KUKA KRL program: EPS_2_251349_CBMH110_A_20251001124302.src

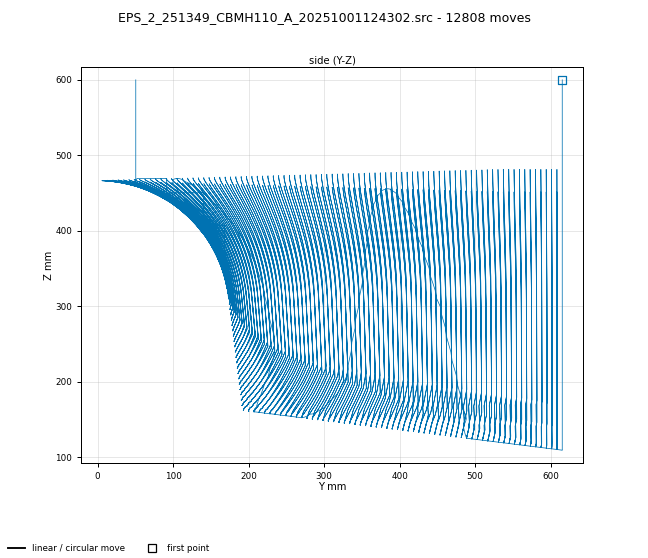
[picture p0: tool path of EPS_2_251349_CBMH110_A_20251001124302.src, 12808 of 12810 moves have a stored position in this frame; points joined in program order, loops and branches not executed]
&ACCESS RVP
&REL 4
&COMMENT QRS 19112012
&PARAM EDITMASK = *
DEF PART()
EXT BAS (BAS_COMMAND :IN,REAL :IN )
INT I
BAS (#INITMOV,0 )

;KUKA QRS Post kuka4.cps  Date:22-06-2017 !

File_ID=2860

QRS_PRE_INIT()

;Init var - Until changes are made in qrs_pre_init
Outlet_Square_prg=0
Inlet_1_Square_prg=0
Inlet_2_Square_prg=0
Inlet_3_Square_prg=0
Inlet_4_Square_prg=0
Inlet_5_Square_prg=0

Outlet_1={X 0.000, Y 534.640, Z 332.000, B 0.000, E1 0.000 }
Inlet_1={X 0.000, Y 536.830, Z 302.000, B 0.000, E1 180.000 }
Outlet_1_type=299
Inlet_1_type=299
;QRS#1=Sidecore dimensions
;QRS#2=300-12" PVC SDR 35
;QRS#3=300-12" PVC SDR 35
;QRS#4=
;QRS#5=
;QRS#6=
;QRS#7=
;QRS#8=
;QRS#9=16M PSX
;QRS#10=16M PSX
;QRS#11=
;QRS#12=
;QRS#13=
;QRS#14=
;QRS#15=
;QRS#16=1220x127x762 2,5'
;QRS#17=EPS Height
;QRS#18=481,5
;QRS#19=*
;QRS#20= UPDATED VERSION 22-06-2017
;QRS#21=*
Outlet_Square=0150
Inlet_1_Square=0150
Inlet_2_Square=0
Inlet_3_Square=0
Inlet_4_Square=0
Inlet_5_Square=0
Mill_Square=1
Outlet_Square_Prg=206
Inlet_1_Square_prg=206

QRS_INIT()

$ADVANCE=5

; T1
PTP {E1 173.632,E2 173.632}
PTP {X 0,Y 615.481,A -85,B 0,C 180,E1 173.632,E2 173.632,E3 0,E4 0,E5 0,E6 0}
QRS_SPEED_INIT()
LIN {X 0,Y 615.481,Z 600,A -85,B 0,C 180,E1 173.632,E2 173.632,E3 0,E4 0,E5 0,E6 0} C_VEL
LIN {X 0,Y 615.481,Z 119.502,A -85,B 0,C 180,E1 173.632,E2 173.632} C_VEL
LIN {X 0,Y 615.481,Z 111.323,A -85,B 0,C 180,E1 173.632,E2 173.632} C_VEL
LIN {X 0,Y 615.461,Z 109.323,A -85,B 0,C 180,E1 173.445,E2 173.445} C_VEL
LIN {X 0,Y 615.458,Z 109.322,A -85,B 0,C 180,E1 171.463,E2 171.463} C_VEL
LIN {X 0,Y 615.439,Z 109.32,A -85,B 0,C 180,E1 169.137,E2 169.137} C_VEL
LIN {X 0,Y 615.448,Z 109.318,A -85,B 0,C 180,E1 166.798,E2 166.798} C_VEL
LIN {X 0,Y 615.49,Z 109.326,A -85,B 0,C 180,E1 164.095,E2 164.095} C_VEL
LIN {X 0,Y 615.436,Z 109.321,A -85,B 0,C 180,E1 161.352,E2 161.352} C_VEL
LIN {X 0,Y 615.487,Z 109.316,A -85,B 0,C 180,E1 158.568,E2 158.568} C_VEL
LIN {X 0,Y 615.441,Z 109.322,A -85,B 0,C 180,E1 155.726,E2 155.726} C_VEL
LIN {X 0,Y 615.431,Z 109.322,A -85,B 0,C 180,E1 153.553,E2 153.553} C_VEL
LIN {X 0,Y 615.434,Z 109.32,A -85,B 0,C 180,E1 151.339,E2 151.339} C_VEL
LIN {X 0,Y 615.469,Z 109.318,A -85,B 0,C 180,E1 148.917,E2 148.917} C_VEL
LIN {X 0,Y 615.437,Z 109.323,A -85,B 0,C 180,E1 145.975,E2 145.975} C_VEL
LIN {X 0,Y 615.429,Z 109.321,A -85,B 0,C 180,E1 143.571,E2 143.571} C_VEL
LIN {X 0,Y 615.49,Z 109.319,A -85,B 0,C 180,E1 140.938,E2 140.938} C_VEL
LIN {X 0,Y 615.465,Z 109.324,A -85,B 0,C 180,E1 138.524,E2 138.524} C_VEL
LIN {X 0,Y 615.424,Z 109.323,A -85,B 0,C 180,E1 136.009,E2 136.009} C_VEL
LIN {X 0,Y 615.422,Z 109.323,A -85,B 0,C 180,E1 133.991,E2 133.991} C_VEL
LIN {X 0,Y 615.447,Z 109.322,A -85,B 0,C 180,E1 131.477,E2 131.477} C_VEL
LIN {X 0,Y 615.479,Z 109.325,A -85,B 0,C 180,E1 128.905,E2 128.905} C_VEL
LIN {X 0,Y 615.425,Z 109.324,A -85,B 0,C 180,E1 126.429,E2 126.429} C_VEL
LIN {X 0,Y 615.459,Z 109.323,A -85,B 0,C 180,E1 123.53,E2 123.53} C_VEL
LIN {X 0,Y 615.45,Z 109.325,A -85,B 0,C 180,E1 120.922,E2 120.922} C_VEL
LIN {X 0,Y 615.414,Z 109.325,A -85,B 0,C 180,E1 118.437,E2 118.437} C_VEL
LIN {X 0,Y 615.413,Z 109.325,A -85,B 0,C 180,E1 116.448,E2 116.448} C_VEL
LIN {X 0,Y 615.432,Z 109.325,A -85,B 0,C 180,E1 113.996,E2 113.996} C_VEL
LIN {X 0,Y 615.418,Z 109.417,A -85,B 0,C 180,E1 112.258,E2 112.258} C_VEL
LIN {X 0,Y 615.49,Z 129.208,A -85,B 0,C 180,E1 109.685,E2 109.685} C_VEL
LIN {X 0,Y 615.468,Z 140.793,A -85,B 0,C 180,E1 108.199,E2 108.199} C_VEL
LIN {X 0,Y 615.481,Z 305.586,A -85,B 0,C 180,E1 106.196,E2 106.196} C_VEL
LIN {X 0,Y 615.497,Z 321.615,A -85,B 0,C 180,E1 105.862,E2 105.862} C_VEL
LIN {X 0,Y 615.488,Z 336.977,A -85,B 0,C 180,E1 105.396,E2 105.396} C_VEL
LIN {X 0,Y 615.483,Z 351.662,A -85,B 0,C 180,E1 104.803,E2 104.803} C_VEL
LIN {X 0,Y 615.492,Z 365.63,A -85,B 0,C 180,E1 104.09,E2 104.09} C_VEL
LIN {X 0,Y 615.498,Z 378.49,A -85,B 0,C 180,E1 103.285,E2 103.285} C_VEL
LIN {X 0,Y 615.496,Z 390.743,A -85,B 0,C 180,E1 102.363,E2 102.363} C_VEL
LIN {X 0,Y 615.498,Z 401.897,A -85,B 0,C 180,E1 101.36,E2 101.36} C_VEL
LIN {X 0,Y 615.497,Z 412.703,A -85,B 0,C 180,E1 100.194,E2 100.194} C_VEL
LIN {X 0,Y 615.495,Z 421.684,A -85,B 0,C 180,E1 99.033,E2 99.033} C_VEL
LIN {X 0,Y 615.493,Z 429.118,A -85,B 0,C 180,E1 97.876,E2 97.876} C_VEL
LIN {X 0,Y 615.492,Z 436.052,A -85,B 0,C 180,E1 96.557,E2 96.557} C_VEL
LIN {X 0,Y 615.489,Z 441.498,A -85,B 0,C 180,E1 95.241,E2 95.241} C_VEL
LIN {X 0,Y 615.495,Z 445.619,A -85,B 0,C 180,E1 93.928,E2 93.928} C_VEL
LIN {X 0,Y 615.493,Z 448.525,A -85,B 0,C 180,E1 92.618,E2 92.618} C_VEL
LIN {X 0,Y 615.491,Z 450.276,A -85,B 0,C 180,E1 91.309,E2 91.309} C_VEL
LIN {X 0,Y 615.492,Z 450.884,A -85,B 0,C 180,E1 90,E2 90} C_VEL
LIN {X 0,Y 615.493,Z 450.338,A -85,B 0,C 180,E1 88.691,E2 88.691} C_VEL
LIN {X 0,Y 615.496,Z 448.674,A -85,B 0,C 180,E1 87.382,E2 87.382} C_VEL
LIN {X 0,Y 615.494,Z 445.861,A -85,B 0,C 180,E1 86.071,E2 86.071} C_VEL
LIN {X 0,Y 615.489,Z 441.835,A -85,B 0,C 180,E1 84.759,E2 84.759} C_VEL
LIN {X 0,Y 615.491,Z 436.378,A -85,B 0,C 180,E1 83.42,E2 83.42} C_VEL
LIN {X 0,Y 615.494,Z 429.66,A -85,B 0,C 180,E1 82.124,E2 82.124} C_VEL
LIN {X 0,Y 615.491,Z 421.144,A -85,B 0,C 180,E1 80.801,E2 80.801} C_VEL
LIN {X 0,Y 615.494,Z 412.066,A -85,B 0,C 180,E1 79.639,E2 79.639} C_VEL
LIN {X 0,Y 615.493,Z 402.791,A -85,B 0,C 180,E1 78.64,E2 78.64} C_VEL
LIN {X 0,Y 615.496,Z 390.821,A -85,B 0,C 180,E1 77.554,E2 77.554} C_VEL
LIN {X 0,Y 615.497,Z 378.58,A -85,B 0,C 180,E1 76.631,E2 76.631} C_VEL
LIN {X 0,Y 615.496,Z 365.88,A -85,B 0,C 180,E1 75.834,E2 75.834} C_VEL
LIN {X 0,Y 615.481,Z 351.779,A -85,B 0,C 180,E1 75.112,E2 75.112} C_VEL
LIN {X 0,Y 615.491,Z 337.119,A -85,B 0,C 180,E1 74.52,E2 74.52} C_VEL
LIN {X 0,Y 615.495,Z 322.175,A -85,B 0,C 180,E1 74.062,E2 74.062} C_VEL
LIN {X 0,Y 615.485,Z 306.977,A -85,B 0,C 180,E1 73.738,E2 73.738} C_VEL
LIN {X 0,Y 615.456,Z 258.405,A -85,B 0,C 180,E1 73.135,E2 73.135} C_VEL
LIN {X 0,Y 615.462,Z 140.874,A -85,B 0,C 180,E1 71.721,E2 71.721} C_VEL
LIN {X 0,Y 615.463,Z 120.461,A -85,B 0,C 180,E1 69.093,E2 69.093} C_VEL
LIN {X 0,Y 615.424,Z 109.324,A -85,B 0,C 180,E1 67.636,E2 67.636} C_VEL
LIN {X 0,Y 615.424,Z 109.324,A -85,B 0,C 180,E1 65.725,E2 65.725} C_VEL
LIN {X 0,Y 615.417,Z 109.324,A -85,B 0,C 180,E1 63.552,E2 63.552} C_VEL
LIN {X 0,Y 615.485,Z 109.328,A -85,B 0,C 180,E1 60.593,E2 60.593} C_VEL
LIN {X 0,Y 615.45,Z 109.325,A -85,B 0,C 180,E1 58.312,E2 58.312} C_VEL
LIN {X 0,Y 615.418,Z 109.325,A -85,B 0,C 180,E1 55.973,E2 55.973} C_VEL
LIN {X 0,Y 615.462,Z 109.325,A -85,B 0,C 180,E1 53.067,E2 53.067} C_VEL
LIN {X 0,Y 615.421,Z 109.325,A -85,B 0,C 180,E1 50.244,E2 50.244} C_VEL
LIN {X 0,Y 615.414,Z 109.325,A -85,B 0,C 180,E1 47.928,E2 47.928} C_VEL
LIN {X 0,Y 615.416,Z 109.325,A -85,B 0,C 180,E1 45.844,E2 45.844} C_VEL
LIN {X 0,Y 615.478,Z 109.325,A -85,B 0,C 180,E1 43.246,E2 43.246} C_VEL
LIN {X 0,Y 615.439,Z 109.323,A -85,B 0,C 180,E1 40.61,E2 40.61} C_VEL
LIN {X 0,Y 615.466,Z 109.322,A -85,B 0,C 180,E1 38.906,E2 38.906} C_VEL
LIN {X 0,Y 615.424,Z 109.323,A -85,B 0,C 180,E1 36.429,E2 36.429} C_VEL
LIN {X 0,Y 615.474,Z 109.326,A -85,B 0,C 180,E1 33.532,E2 33.532} C_VEL
LIN {X 0,Y 615.449,Z 109.321,A -85,B 0,C 180,E1 30.922,E2 30.922} C_VEL
LIN {X 0,Y 615.426,Z 109.322,A -85,B 0,C 180,E1 28.439,E2 28.439} C_VEL
LIN {X 0,Y 615.498,Z 109.324,A -85,B 0,C 180,E1 25.57,E2 25.57} C_VEL
LIN {X 0,Y 615.434,Z 109.32,A -85,B 0,C 180,E1 22.847,E2 22.847} C_VEL
LIN {X 0,Y 615.431,Z 109.322,A -85,B 0,C 180,E1 20.542,E2 20.542} C_VEL
LIN {X 0,Y 615.483,Z 109.324,A -85,B 0,C 180,E1 17.957,E2 17.957} C_VEL
LIN {X 0,Y 615.449,Z 109.319,A -85,B 0,C 180,E1 15.227,E2 15.227} C_VEL
LIN {X 0,Y 615.445,Z 109.319,A -85,B 0,C 180,E1 13.202,E2 13.202} C_VEL
LIN {X 0,Y 615.435,Z 109.321,A -85,B 0,C 180,E1 10.861,E2 10.861} C_VEL
LIN {X 0,Y 615.452,Z 109.323,A -85,B 0,C 180,E1 8.537,E2 8.537} C_VEL
LIN {X 0,Y 615.499,Z 109.316,A -85,B 0,C 180,E1 5.899,E2 5.899} C_VEL
LIN {X 0,Y 615.44,Z 109.319,A -85,B 0,C 180,E1 3.273,E2 3.273} C_VEL
LIN {X 0,Y 615.441,Z 109.318,A -85,B 0,C 180,E1 1.309,E2 1.309} C_VEL
LIN {X 0,Y 615.465,Z 109.323,A -85,B 0,C 180,E1 -1.309,E2 -1.309} C_VEL
LIN {X 0,Y 615.486,Z 109.316,A -85,B 0,C 180,E1 -3.928,E2 -3.928} C_VEL
LIN {X 0,Y 615.444,Z 109.318,A -85,B 0,C 180,E1 -6.557,E2 -6.557} C_VEL
LIN {X 0,Y 615.478,Z 109.324,A -85,B 0,C 180,E1 -9.199,E2 -9.199} C_VEL
LIN {X 0,Y 615.48,Z 109.313,A -85,B 0,C 180,E1 -11.861,E2 -11.861} C_VEL
LIN {X 0,Y 615.448,Z 109.319,A -85,B 0,C 180,E1 -14.55,E2 -14.55} C_VEL
LIN {X 0,Y 615.494,Z 109.322,A -85,B 0,C 180,E1 -17.27,E2 -17.27} C_VEL
LIN {X 0,Y 615.457,Z 109.315,A -85,B 0,C 180,E1 -20.034,E2 -20.034} C_VEL
LIN {X 0,Y 615.452,Z 109.318,A -85,B 0,C 180,E1 -22.337,E2 -22.337} C_VEL
LIN {X 0,Y 615.493,Z 109.324,A -85,B 0,C 180,E1 -24.991,E2 -24.991} C_VEL
LIN {X 0,Y 615.457,Z 109.315,A -85,B 0,C 180,E1 -27.917,E2 -27.917} C_VEL
LIN {X 0,Y 615.455,Z 109.318,A -85,B 0,C 180,E1 -30.162,E2 -30.162} C_VEL
LIN {X 0,Y 615.475,Z 109.322,A -85,B 0,C 180,E1 -32.458,E2 -32.458} C_VEL
LIN {X 0,Y 615.493,Z 109.32,A -85,B 0,C 180,E1 -34.815,E2 -34.815} C_VEL
LIN {X 0,Y 615.49,Z 109.309,A -85,B 0,C 180,E1 -37.242,E2 -37.242} C_VEL
LIN {X 0,Y 615.458,Z 109.316,A -85,B 0,C 180,E1 -39.752,E2 -39.752} C_VEL
LIN {X 0,Y 615.492,Z 109.324,A -85,B 0,C 180,E1 -42.353,E2 -42.353} C_VEL
LIN {X 0,Y 615.492,Z 109.308,A -85,B 0,C 180,E1 -45.068,E2 -45.068} C_VEL
LIN {X 0,Y 615.47,Z 109.321,A -85,B 0,C 180,E1 -47.922,E2 -47.922} C_VEL
LIN {X 0,Y 615.493,Z 109.308,A -85,B 0,C 180,E1 -50.937,E2 -50.937} C_VEL
LIN {X 0,Y 615.464,Z 109.318,A -85,B 0,C 180,E1 -53.573,E2 -53.573} C_VEL
LIN {X 0,Y 615.489,Z 109.314,A -85,B 0,C 180,E1 -56.466,E2 -56.466} C_VEL
LIN {X 0,Y 615.47,Z 109.312,A -85,B 0,C 180,E1 -59.079,E2 -59.079} C_VEL
LIN {X 0,Y 615.475,Z 109.32,A -85,B 0,C 180,E1 -61.552,E2 -61.552} C_VEL
LIN {X 0,Y 615.488,Z 109.31,A -85,B 0,C 180,E1 -64.431,E2 -64.431} C_VEL
LIN {X 0,Y 615.473,Z 109.433,A -85,B 0,C 180,E1 -64.935,E2 -64.935} C_VEL
LIN {X 0,Y 615.485,Z 133.182,A -85,B 0,C 180,E1 -67.655,E2 -67.655} C_VEL
LIN {X 0,Y 615.498,Z 158.435,A -85,B 0,C 180,E1 -70.489,E2 -70.489} C_VEL
LIN {X 0,Y 615.487,Z 170.026,A -85,B 0,C 180,E1 -71.762,E2 -71.762} C_VEL
LIN {X 0,Y 615.483,Z 336.208,A -85,B 0,C 180,E1 -73.769,E2 -73.769} C_VEL
LIN {X 0,Y 615.496,Z 351.709,A -85,B 0,C 180,E1 -74.095,E2 -74.095} C_VEL
LIN {X 0,Y 615.489,Z 367.048,A -85,B 0,C 180,E1 -74.562,E2 -74.562} C_VEL
LIN {X 0,Y 615.484,Z 380.751,A -85,B 0,C 180,E1 -75.113,E2 -75.113} C_VEL
LIN {X 0,Y 615.493,Z 395.045,A -85,B 0,C 180,E1 -75.833,E2 -75.833} C_VEL
LIN {X 0,Y 615.497,Z 407.897,A -85,B 0,C 180,E1 -76.631,E2 -76.631} C_VEL
LIN {X 0,Y 615.495,Z 420.254,A -85,B 0,C 180,E1 -77.554,E2 -77.554} C_VEL
LIN {X 0,Y 615.496,Z 430.606,A -85,B 0,C 180,E1 -78.473,E2 -78.473} C_VEL
LIN {X 0,Y 615.494,Z 440.183,A -85,B 0,C 180,E1 -79.473,E2 -79.473} C_VEL
LIN {X 0,Y 615.494,Z 449.577,A -85,B 0,C 180,E1 -80.636,E2 -80.636} C_VEL
LIN {X 0,Y 615.494,Z 457.38,A -85,B 0,C 180,E1 -81.794,E2 -81.794} C_VEL
LIN {X 0,Y 615.494,Z 464.609,A -85,B 0,C 180,E1 -83.102,E2 -83.102} C_VEL
LIN {X 0,Y 615.499,Z 470.436,A -85,B 0,C 180,E1 -84.43,E2 -84.43} C_VEL
LIN {X 0,Y 615.491,Z 473.86,A -85,B 0,C 180,E1 -85.415,E2 -85.415} C_VEL
LIN {X 0,Y 615.493,Z 477.318,A -85,B 0,C 180,E1 -86.727,E2 -86.727} C_VEL
LIN {X 0,Y 615.5,Z 479.593,A -85,B 0,C 180,E1 -88.037,E2 -88.037} C_VEL
LIN {X 0,Y 615.491,Z 480.741,A -85,B 0,C 180,E1 -89.346,E2 -89.346} C_VEL
LIN {X 0,Y 615.491,Z 480.741,A -85,B 0,C 180,E1 -90.654,E2 -90.654} C_VEL
LIN {X 0,Y 615.5,Z 479.593,A -85,B 0,C 180,E1 -91.963,E2 -91.963} C_VEL
LIN {X 0,Y 615.493,Z 477.318,A -85,B 0,C 180,E1 -93.273,E2 -93.273} C_VEL
LIN {X 0,Y 615.491,Z 473.86,A -85,B 0,C 180,E1 -94.585,E2 -94.585} C_VEL
LIN {X 0,Y 615.499,Z 469.142,A -85,B 0,C 180,E1 -95.898,E2 -95.898} C_VEL
LIN {X 0,Y 615.492,Z 463.03,A -85,B 0,C 180,E1 -97.216,E2 -97.216} C_VEL
LIN {X 0,Y 615.493,Z 455.332,A -85,B 0,C 180,E1 -98.537,E2 -98.537} C_VEL
LIN {X 0,Y 615.495,Z 447.113,A -85,B 0,C 180,E1 -99.696,E2 -99.696} C_VEL
LIN {X 0,Y 615.496,Z 436.899,A -85,B 0,C 180,E1 -100.892,E2 -100.892} C_VEL
LIN {X 0,Y 615.496,Z 427.067,A -85,B 0,C 180,E1 -101.861,E2 -101.861} C_VEL
LIN {X 0,Y 615.497,Z 414.947,A -85,B 0,C 180,E1 -102.865,E2 -102.865} C_VEL
LIN {X 0,Y 615.498,Z 402.797,A -85,B 0,C 180,E1 -103.706,E2 -103.706} C_VEL
LIN {X 0,Y 615.477,Z 389.378,A -85,B 0,C 180,E1 -104.473,E2 -104.473} C_VEL
LIN {X 0,Y 615.497,Z 374.846,A -85,B 0,C 180,E1 -105.141,E2 -105.141} C_VEL
LIN {X 0,Y 615.494,Z 360.614,A -85,B 0,C 180,E1 -105.65,E2 -105.65} C_VEL
LIN {X 0,Y 615.498,Z 346.141,A -85,B 0,C 180,E1 -106.036,E2 -106.036} C_VEL
LIN {X 0,Y 615.484,Z 331.616,A -85,B 0,C 180,E1 -106.297,E2 -106.297} C_VEL
LIN {X 0,Y 615.489,Z 169.742,A -85,B 0,C 180,E1 -108.258,E2 -108.258} C_VEL
LIN {X 0,Y 615.49,Z 144.391,A -85,B 0,C 180,E1 -111.081,E2 -111.081} C_VEL
LIN {X 0,Y 615.482,Z 120.569,A -85,B 0,C 180,E1 -113.782,E2 -113.782} C_VEL
LIN {X 0,Y 615.474,Z 109.311,A -85,B 0,C 180,E1 -115.1,E2 -115.1} C_VEL
LIN {X 0,Y 615.488,Z 109.319,A -85,B 0,C 180,E1 -117.915,E2 -117.915} C_VEL
LIN {X 0,Y 615.49,Z 109.325,A -85,B 0,C 180,E1 -120.16,E2 -120.16} C_VEL
LIN {X 0,Y 615.469,Z 109.319,A -85,B 0,C 180,E1 -122.459,E2 -122.459} C_VEL
LIN {X 0,Y 615.469,Z 109.313,A -85,B 0,C 180,E1 -124.816,E2 -124.816} C_VEL
LIN {X 0,Y 615.494,Z 109.309,A -85,B 0,C 180,E1 -127.242,E2 -127.242} C_VEL
LIN {X 0,Y 615.476,Z 109.321,A -85,B 0,C 180,E1 -130.088,E2 -130.088} C_VEL
LIN {X 0,Y 615.462,Z 109.317,A -85,B 0,C 180,E1 -132.355,E2 -132.355} C_VEL
LIN {X 0,Y 615.492,Z 109.31,A -85,B 0,C 180,E1 -135.068,E2 -135.068} C_VEL
LIN {X 0,Y 615.471,Z 109.321,A -85,B 0,C 180,E1 -137.922,E2 -137.922} C_VEL
LIN {X 0,Y 615.458,Z 109.316,A -85,B 0,C 180,E1 -140.248,E2 -140.248} C_VEL
LIN {X 0,Y 615.492,Z 109.315,A -85,B 0,C 180,E1 -143.063,E2 -143.063} C_VEL
LIN {X 0,Y 615.458,Z 109.318,A -85,B 0,C 180,E1 -145.976,E2 -145.976} C_VEL
LIN {X 0,Y 615.462,Z 109.314,A -85,B 0,C 180,E1 -148.313,E2 -148.313} C_VEL
LIN {X 0,Y 615.486,Z 109.324,A -85,B 0,C 180,E1 -151.342,E2 -151.342} C_VEL
LIN {X 0,Y 615.463,Z 109.321,A -85,B 0,C 180,E1 -153.555,E2 -153.555} C_VEL
LIN {X 0,Y 615.457,Z 109.315,A -85,B 0,C 180,E1 -155.999,E2 -155.999} C_VEL
LIN {X 0,Y 615.496,Z 109.312,A -85,B 0,C 180,E1 -158.569,E2 -158.569} C_VEL
LIN {X 0,Y 615.457,Z 109.32,A -85,B 0,C 180,E1 -161.404,E2 -161.404} C_VEL
LIN {X 0,Y 615.472,Z 109.313,A -85,B 0,C 180,E1 -164.094,E2 -164.094} C_VEL
LIN {X 0,Y 615.496,Z 109.325,A -85,B 0,C 180,E1 -166.799,E2 -166.799} C_VEL
LIN {X 0,Y 615.448,Z 109.318,A -85,B 0,C 180,E1 -169.472,E2 -169.472} C_VEL
LIN {X 0,Y 615.484,Z 109.314,A -85,B 0,C 180,E1 -172.124,E2 -172.124} C_VEL
LIN {X 0,Y 615.475,Z 109.323,A -85,B 0,C 180,E1 -174.759,E2 -174.759} C_VEL
LIN {X 0,Y 615.446,Z 109.318,A -85,B 0,C 180,E1 -177.382,E2 -177.382} C_VEL
LIN {X 0,Y 615.487,Z 109.315,A -85,B 0,C 180,E1 -180,E2 -180} C_VEL
LIN {X 0,Y 615.466,Z 109.323,A -85,B 0,C 180,E1 -182.618,E2 -182.618} C_VEL
LIN {X 0,Y 615.442,Z 109.318,A -85,B 0,C 180,E1 -185.242,E2 -185.242} C_VEL
LIN {X 0,Y 615.461,Z 109.323,A -85,B 0,C 180,E1 -186.555,E2 -186.555} C_VEL
LIN {X 0,Y 614.772,Z 109.465,A -85,B 0,C 180,E1 -187.101,E2 -187.101} C_VEL
LIN {X 0,Y 611.925,Z 109.887,A -85,B 0,C 180,E1 -187.987,E2 -187.987} C_VEL
LIN {X 0,Y 609.539,Z 110.191,A -85,B 0,C 180,E1 -188.699,E2 -188.699} C_VEL
LIN {X 0,Y 608.519,Z 110.306,A -85,B 0,C 180,E1 -189.249,E2 -189.249} C_VEL
LIN {X 0,Y 608.437,Z 110.315,A -85,B 0,C 180,E1 -189.435,E2 -189.435} C_VEL
LIN {X 0,Y 608.46,Z 110.321,A -85,B 0,C 180,E1 -192,E2 -192} C_VEL
LIN {X 0,Y 608.409,Z 110.319,A -85,B 0,C 180,E1 -194.722,E2 -194.722} C_VEL
LIN {X 0,Y 608.417,Z 110.317,A -85,B 0,C 180,E1 -196.785,E2 -196.785} C_VEL
LIN {X 0,Y 608.439,Z 110.32,A -85,B 0,C 180,E1 -199.571,E2 -199.571} C_VEL
LIN {X 0,Y 608.432,Z 110.316,A -85,B 0,C 180,E1 -202.469,E2 -202.469} C_VEL
LIN {X 0,Y 608.418,Z 110.317,A -85,B 0,C 180,E1 -204.573,E2 -204.573} C_VEL
LIN {X 0,Y 608.462,Z 110.315,A -85,B 0,C 180,E1 -207.204,E2 -207.204} C_VEL
LIN {X 0,Y 608.424,Z 110.32,A -85,B 0,C 180,E1 -209.964,E2 -209.964} C_VEL
LIN {X 0,Y 608.415,Z 110.317,A -85,B 0,C 180,E1 -212.515,E2 -212.515} C_VEL
LIN {X 0,Y 608.417,Z 110.319,A -85,B 0,C 180,E1 -214.901,E2 -214.901} C_VEL
LIN {X 0,Y 608.438,Z 110.318,A -85,B 0,C 180,E1 -217.749,E2 -217.749} C_VEL
LIN {X 0,Y 608.403,Z 110.319,A -85,B 0,C 180,E1 -220.323,E2 -220.323} C_VEL
LIN {X 0,Y 608.444,Z 110.32,A -85,B 0,C 180,E1 -222.961,E2 -222.961} C_VEL
LIN {X 0,Y 608.408,Z 110.32,A -85,B 0,C 180,E1 -225.741,E2 -225.741} C_VEL
LIN {X 0,Y 608.405,Z 110.319,A -85,B 0,C 180,E1 -227.934,E2 -227.934} C_VEL
LIN {X 0,Y 608.435,Z 110.321,A -85,B 0,C 180,E1 -230.707,E2 -230.707} C_VEL
LIN {X 0,Y 608.442,Z 110.321,A -85,B 0,C 180,E1 -233.084,E2 -233.084} C_VEL
LIN {X 0,Y 608.42,Z 110.318,A -85,B 0,C 180,E1 -235.527,E2 -235.527} C_VEL
LIN {X 0,Y 608.411,Z 110.318,A -85,B 0,C 180,E1 -237.902,E2 -237.902} C_VEL
LIN {X 0,Y 608.426,Z 110.319,A -85,B 0,C 180,E1 -240.218,E2 -240.218} C_VEL
LIN {X 0,Y 608.461,Z 110.319,A -85,B 0,C 180,E1 -242.796,E2 -242.796} C_VEL
LIN {X 0,Y 608.403,Z 110.319,A -85,B 0,C 180,E1 -245.427,E2 -245.427} C_VEL
LIN {X 0,Y 608.387,Z 110.328,A -85,B 0,C 180,E1 -247.591,E2 -247.591} C_VEL
LIN {X 0,Y 608.554,Z 123.245,A -85,B 0,C 180,E1 -249.3,E2 -249.3} C_VEL
LIN {X 0,Y 608.523,Z 140.819,A -85,B 0,C 180,E1 -251.586,E2 -251.586} C_VEL
LIN {X 0,Y 608.745,Z 144.647,A -85,B 0,C 180,E1 -251.654,E2 -251.654} C_VEL
LIN {X 0,Y 608.682,Z 305.623,A -85,B 0,C 180,E1 -253.618,E2 -253.618} C_VEL
LIN {X 0,Y 608.667,Z 321.637,A -85,B 0,C 180,E1 -253.955,E2 -253.955} C_VEL
LIN {X 0,Y 608.62,Z 336.992,A -85,B 0,C 180,E1 -254.426,E2 -254.426} C_VEL
LIN {X 0,Y 608.589,Z 351.673,A -85,B 0,C 180,E1 -255.026,E2 -255.026} C_VEL
LIN {X 0,Y 608.57,Z 365.44,A -85,B 0,C 180,E1 -255.735,E2 -255.735} C_VEL
LIN {X 0,Y 608.548,Z 378.544,A -85,B 0,C 180,E1 -256.56,E2 -256.56} C_VEL
LIN {X 0,Y 608.505,Z 390.84,A -85,B 0,C 180,E1 -257.493,E2 -257.493} C_VEL
LIN {X 0,Y 608.498,Z 402.05,A -85,B 0,C 180,E1 -258.508,E2 -258.508} C_VEL
LIN {X 0,Y 608.477,Z 412.935,A -85,B 0,C 180,E1 -259.687,E2 -259.687} C_VEL
LIN {X 0,Y 608.469,Z 421.984,A -85,B 0,C 180,E1 -260.862,E2 -260.862} C_VEL
LIN {X 0,Y 608.456,Z 429.48,A -85,B 0,C 180,E1 -262.033,E2 -262.033} C_VEL
LIN {X 0,Y 608.445,Z 436.629,A -85,B 0,C 180,E1 -263.397,E2 -263.397} C_VEL
LIN {X 0,Y 608.435,Z 441.993,A -85,B 0,C 180,E1 -264.698,E2 -264.698} C_VEL
LIN {X 0,Y 608.432,Z 446.167,A -85,B 0,C 180,E1 -266.026,E2 -266.026} C_VEL
LIN {X 0,Y 608.421,Z 449.11,A -85,B 0,C 180,E1 -267.352,E2 -267.352} C_VEL
LIN {X 0,Y 608.444,Z 450.88,A -85,B 0,C 180,E1 -268.676,E2 -268.676} C_VEL
LIN {X 0,Y 608.432,Z 451.495,A -85,B 0,C 180,E1 -270,E2 -270} C_VEL
LIN {X 0,Y 608.445,Z 450.944,A -85,B 0,C 180,E1 -271.324,E2 -271.324} C_VEL
LIN {X 0,Y 608.424,Z 449.259,A -85,B 0,C 180,E1 -272.648,E2 -272.648} C_VEL
LIN {X 0,Y 608.431,Z 446.408,A -85,B 0,C 180,E1 -273.974,E2 -273.974} C_VEL
LIN {X 0,Y 608.435,Z 442.328,A -85,B 0,C 180,E1 -275.302,E2 -275.302} C_VEL
LIN {X 0,Y 608.446,Z 436.921,A -85,B 0,C 180,E1 -276.633,E2 -276.633} C_VEL
LIN {X 0,Y 608.457,Z 430.022,A -85,B 0,C 180,E1 -277.967,E2 -277.967} C_VEL
LIN {X 0,Y 608.466,Z 422.591,A -85,B 0,C 180,E1 -279.138,E2 -279.138} C_VEL
LIN {X 0,Y 608.476,Z 413.662,A -85,B 0,C 180,E1 -280.313,E2 -280.313} C_VEL
LIN {X 0,Y 608.495,Z 402.946,A -85,B 0,C 180,E1 -281.492,E2 -281.492} C_VEL
LIN {X 0,Y 608.513,Z 390.904,A -85,B 0,C 180,E1 -282.591,E2 -282.591} C_VEL
LIN {X 0,Y 608.543,Z 378.616,A -85,B 0,C 180,E1 -283.525,E2 -283.525} C_VEL
LIN {X 0,Y 608.585,Z 365.673,A -85,B 0,C 180,E1 -284.342,E2 -284.342} C_VEL
LIN {X 0,Y 608.584,Z 351.767,A -85,B 0,C 180,E1 -285.06,E2 -285.06} C_VEL
LIN {X 0,Y 608.645,Z 337.102,A -85,B 0,C 180,E1 -285.659,E2 -285.659} C_VEL
LIN {X 0,Y 608.661,Z 321.545,A -85,B 0,C 180,E1 -286.138,E2 -286.138} C_VEL
LIN {X 0,Y 608.676,Z 305.808,A -85,B 0,C 180,E1 -286.47,E2 -286.47} C_VEL
LIN {X 0,Y 608.721,Z 142.059,A -85,B 0,C 180,E1 -288.469,E2 -288.469} C_VEL
LIN {X 0,Y 608.515,Z 140.891,A -85,B 0,C 180,E1 -288.495,E2 -288.495} C_VEL
LIN {X 0,Y 608.552,Z 120.459,A -85,B 0,C 180,E1 -291.155,E2 -291.155} C_VEL
LIN {X 0,Y 608.395,Z 110.322,A -85,B 0,C 180,E1 -292.509,E2 -292.509} C_VEL
LIN {X 0,Y 608.408,Z 110.319,A -85,B 0,C 180,E1 -294.573,E2 -294.573} C_VEL
LIN {X 0,Y 608.459,Z 110.318,A -85,B 0,C 180,E1 -297.203,E2 -297.203} C_VEL
LIN {X 0,Y 608.406,Z 110.32,A -85,B 0,C 180,E1 -299.961,E2 -299.961} C_VEL
LIN {X 0,Y 608.404,Z 110.319,A -85,B 0,C 180,E1 -302.514,E2 -302.514} C_VEL
LIN {X 0,Y 608.407,Z 110.328,A -85,B 0,C 180,E1 -305.28,E2 -305.28} C_VEL
LIN {X 0,Y 608.401,Z 110.321,A -85,B 0,C 180,E1 -307.751,E2 -307.751} C_VEL
LIN {X 0,Y 608.403,Z 110.319,A -85,B 0,C 180,E1 -310.323,E2 -310.323} C_VEL
LIN {X 0,Y 608.439,Z 110.324,A -85,B 0,C 180,E1 -312.961,E2 -312.961} C_VEL
LIN {X 0,Y 608.401,Z 110.319,A -85,B 0,C 180,E1 -315.742,E2 -315.742} C_VEL
LIN {X 0,Y 608.403,Z 110.319,A -85,B 0,C 180,E1 -317.934,E2 -317.934} C_VEL
LIN {X 0,Y 608.434,Z 110.324,A -85,B 0,C 180,E1 -320.707,E2 -320.707} C_VEL
LIN {X 0,Y 608.433,Z 110.319,A -85,B 0,C 180,E1 -323.083,E2 -323.083} C_VEL
LIN {X 0,Y 608.423,Z 110.316,A -85,B 0,C 180,E1 -325.528,E2 -325.528} C_VEL
LIN {X 0,Y 608.422,Z 110.317,A -85,B 0,C 180,E1 -327.903,E2 -327.903} C_VEL
LIN {X 0,Y 608.44,Z 110.319,A -85,B 0,C 180,E1 -330.219,E2 -330.219} C_VEL
LIN {X 0,Y 608.403,Z 110.319,A -85,B 0,C 180,E1 -333.223,E2 -333.223} C_VEL
LIN {X 0,Y 608.415,Z 110.317,A -85,B 0,C 180,E1 -335.427,E2 -335.427} C_VEL
LIN {X 0,Y 608.456,Z 110.322,A -85,B 0,C 180,E1 -338.308,E2 -338.308} C_VEL
LIN {X 0,Y 608.418,Z 110.317,A -85,B 0,C 180,E1 -341.3,E2 -341.3} C_VEL
LIN {X 0,Y 608.445,Z 110.32,A -85,B 0,C 180,E1 -343.906,E2 -343.906} C_VEL
LIN {X 0,Y 608.437,Z 110.316,A -85,B 0,C 180,E1 -346.643,E2 -346.643} C_VEL
LIN {X 0,Y 608.424,Z 110.318,A -85,B 0,C 180,E1 -349.349,E2 -349.349} C_VEL
LIN {X 0,Y 608.477,Z 110.317,A -85,B 0,C 180,E1 -352.033,E2 -352.033} C_VEL
LIN {X 0,Y 608.427,Z 110.316,A -85,B 0,C 180,E1 -354.698,E2 -354.698} C_VEL
LIN {X 0,Y 608.449,Z 110.317,A -85,B 0,C 180,E1 -357.352,E2 -357.352} C_VEL
LIN {X 0,Y 608.477,Z 110.314,A -85,B 0,C 180,E1 -360,E2 -360} C_VEL
LIN {X 0,Y 608.439,Z 110.314,A -85,B 0,C 180,E1 -362.648,E2 -362.648} C_VEL
LIN {X 0,Y 608.453,Z 110.32,A -85,B 0,C 180,E1 -365.302,E2 -365.302} C_VEL
LIN {X 0,Y 608.471,Z 110.312,A -85,B 0,C 180,E1 -367.967,E2 -367.967} C_VEL
LIN {X 0,Y 608.43,Z 110.317,A -85,B 0,C 180,E1 -370.65,E2 -370.65} C_VEL
LIN {X 0,Y 608.467,Z 110.32,A -85,B 0,C 180,E1 -373.356,E2 -373.356} C_VEL
LIN {X 0,Y 608.439,Z 110.314,A -85,B 0,C 180,E1 -376.094,E2 -376.094} C_VEL
LIN {X 0,Y 608.448,Z 110.32,A -85,B 0,C 180,E1 -378.87,E2 -378.87} C_VEL
LIN {X 0,Y 608.463,Z 110.312,A -85,B 0,C 180,E1 -381.692,E2 -381.692} C_VEL
LIN {X 0,Y 608.44,Z 110.319,A -85,B 0,C 180,E1 -384.572,E2 -384.572} C_VEL
LIN {X 0,Y 608.486,Z 110.313,A -85,B 0,C 180,E1 -387.208,E2 -387.208} C_VEL
LIN {X 0,Y 608.426,Z 110.316,A -85,B 0,C 180,E1 -389.964,E2 -389.964} C_VEL
LIN {X 0,Y 608.453,Z 110.32,A -85,B 0,C 180,E1 -392.521,E2 -392.521} C_VEL
LIN {X 0,Y 608.434,Z 110.316,A -85,B 0,C 180,E1 -395.278,E2 -395.278} C_VEL
LIN {X 0,Y 608.453,Z 110.313,A -85,B 0,C 180,E1 -397.747,E2 -397.747} C_VEL
LIN {X 0,Y 608.442,Z 110.322,A -85,B 0,C 180,E1 -400.328,E2 -400.328} C_VEL
LIN {X 0,Y 608.468,Z 110.311,A -85,B 0,C 180,E1 -403.308,E2 -403.308} C_VEL
LIN {X 0,Y 608.458,Z 110.319,A -85,B 0,C 180,E1 -406.129,E2 -406.129} C_VEL
LIN {X 0,Y 608.458,Z 110.314,A -85,B 0,C 180,E1 -408.823,E2 -408.823} C_VEL
LIN {X 0,Y 608.434,Z 110.316,A -85,B 0,C 180,E1 -411.409,E2 -411.409} C_VEL
LIN {X 0,Y 608.448,Z 110.322,A -85,B 0,C 180,E1 -413.954,E2 -413.954} C_VEL
LIN {X 0,Y 608.466,Z 110.316,A -85,B 0,C 180,E1 -416.329,E2 -416.329} C_VEL
LIN {X 0,Y 608.447,Z 110.314,A -85,B 0,C 180,E1 -418.732,E2 -418.732} C_VEL
LIN {X 0,Y 608.461,Z 110.315,A -85,B 0,C 180,E1 -421.382,E2 -421.382} C_VEL
LIN {X 0,Y 608.444,Z 110.323,A -85,B 0,C 180,E1 -423.964,E2 -423.964} C_VEL
LIN {X 0,Y 608.485,Z 110.446,A -85,B 0,C 180,E1 -424.746,E2 -424.746} C_VEL
LIN {X 0,Y 608.657,Z 122.541,A -85,B 0,C 180,E1 -426.163,E2 -426.163} C_VEL
LIN {X 0,Y 608.596,Z 145.951,A -85,B 0,C 180,E1 -428.846,E2 -428.846} C_VEL
LIN {X 0,Y 608.575,Z 170.026,A -85,B 0,C 180,E1 -431.547,E2 -431.547} C_VEL
LIN {X 0,Y 608.71,Z 279.271,A -85,B 0,C 180,E1 -432.877,E2 -432.877} C_VEL
LIN {X 0,Y 608.678,Z 336.207,A -85,B 0,C 180,E1 -433.582,E2 -433.582} C_VEL
LIN {X 0,Y 608.671,Z 351.708,A -85,B 0,C 180,E1 -433.912,E2 -433.912} C_VEL
LIN {X 0,Y 608.631,Z 367.046,A -85,B 0,C 180,E1 -434.384,E2 -434.384} C_VEL
LIN {X 0,Y 608.605,Z 380.755,A -85,B 0,C 180,E1 -434.94,E2 -434.94} C_VEL
LIN {X 0,Y 608.572,Z 394.235,A -85,B 0,C 180,E1 -435.624,E2 -435.624} C_VEL
LIN {X 0,Y 608.554,Z 406.663,A -85,B 0,C 180,E1 -436.39,E2 -436.39} C_VEL
LIN {X 0,Y 608.528,Z 419.282,A -85,B 0,C 180,E1 -437.324,E2 -437.324} C_VEL
LIN {X 0,Y 608.497,Z 430.747,A -85,B 0,C 180,E1 -438.339,E2 -438.339} C_VEL
LIN {X 0,Y 608.475,Z 440.388,A -85,B 0,C 180,E1 -439.35,E2 -439.35} C_VEL
LIN {X 0,Y 608.477,Z 449.853,A -85,B 0,C 180,E1 -440.527,E2 -440.527} C_VEL
LIN {X 0,Y 608.456,Z 457.729,A -85,B 0,C 180,E1 -441.698,E2 -441.698} C_VEL
LIN {X 0,Y 608.439,Z 465.087,A -85,B 0,C 180,E1 -443.034,E2 -443.034} C_VEL
LIN {X 0,Y 608.451,Z 470.923,A -85,B 0,C 180,E1 -444.366,E2 -444.366} C_VEL
LIN {X 0,Y 608.427,Z 474.383,A -85,B 0,C 180,E1 -445.362,E2 -445.362} C_VEL
LIN {X 0,Y 608.421,Z 477.885,A -85,B 0,C 180,E1 -446.689,E2 -446.689} C_VEL
LIN {X 0,Y 608.444,Z 480.191,A -85,B 0,C 180,E1 -448.014,E2 -448.014} C_VEL
LIN {X 0,Y 608.434,Z 481.35,A -85,B 0,C 180,E1 -449.338,E2 -449.338} C_VEL
LIN {X 0,Y 608.434,Z 481.35,A -85,B 0,C 180,E1 -450.662,E2 -450.662} C_VEL
LIN {X 0,Y 608.444,Z 480.191,A -85,B 0,C 180,E1 -451.986,E2 -451.986} C_VEL
LIN {X 0,Y 608.421,Z 477.885,A -85,B 0,C 180,E1 -453.311,E2 -453.311} C_VEL
LIN {X 0,Y 608.427,Z 474.383,A -85,B 0,C 180,E1 -454.638,E2 -454.638} C_VEL
LIN {X 0,Y 608.437,Z 469.608,A -85,B 0,C 180,E1 -455.967,E2 -455.967} C_VEL
LIN {X 0,Y 608.456,Z 463.426,A -85,B 0,C 180,E1 -457.3,E2 -457.3} C_VEL
LIN {X 0,Y 608.467,Z 455.654,A -85,B 0,C 180,E1 -458.636,E2 -458.636} C_VEL
LIN {X 0,Y 608.471,Z 447.37,A -85,B 0,C 180,E1 -459.809,E2 -459.809} C_VEL
LIN {X 0,Y 608.492,Z 436.652,A -85,B 0,C 180,E1 -461.063,E2 -461.063} C_VEL
LIN {X 0,Y 608.522,Z 425.274,A -85,B 0,C 180,E1 -462.168,E2 -462.168} C_VEL
LIN {X 0,Y 608.547,Z 413.854,A -85,B 0,C 180,E1 -463.1,E2 -463.1} C_VEL
LIN {X 0,Y 608.563,Z 401.446,A -85,B 0,C 180,E1 -463.95,E2 -463.95} C_VEL
LIN {X 0,Y 608.561,Z 387.858,A -85,B 0,C 180,E1 -464.718,E2 -464.718} C_VEL
LIN {X 0,Y 608.638,Z 373.79,A -85,B 0,C 180,E1 -465.359,E2 -465.359} C_VEL
LIN {X 0,Y 608.644,Z 359.299,A -85,B 0,C 180,E1 -465.874,E2 -465.874} C_VEL
LIN {X 0,Y 608.686,Z 344.023,A -85,B 0,C 180,E1 -466.269,E2 -466.269} C_VEL
LIN {X 0,Y 608.685,Z 328.103,A -85,B 0,C 180,E1 -466.534,E2 -466.534} C_VEL
LIN {X 0,Y 608.684,Z 170.657,A -85,B 0,C 180,E1 -468.442,E2 -468.442} C_VEL
LIN {X 0,Y 608.541,Z 169.567,A -85,B 0,C 180,E1 -468.495,E2 -468.495} C_VEL
LIN {X 0,Y 608.596,Z 145.951,A -85,B 0,C 180,E1 -471.154,E2 -471.154} C_VEL
LIN {X 0,Y 608.657,Z 122.541,A -85,B 0,C 180,E1 -473.837,E2 -473.837} C_VEL
LIN {X 0,Y 608.485,Z 110.446,A -85,B 0,C 180,E1 -475.254,E2 -475.254} C_VEL
LIN {X 0,Y 608.448,Z 110.315,A -85,B 0,C 180,E1 -477.518,E2 -477.518} C_VEL
LIN {X 0,Y 608.469,Z 110.319,A -85,B 0,C 180,E1 -479.972,E2 -479.972} C_VEL
LIN {X 0,Y 608.452,Z 110.313,A -85,B 0,C 180,E1 -482.88,E2 -482.88} C_VEL
LIN {X 0,Y 608.437,Z 110.316,A -85,B 0,C 180,E1 -485.278,E2 -485.278} C_VEL
LIN {X 0,Y 608.469,Z 110.319,A -85,B 0,C 180,E1 -487.746,E2 -487.746} C_VEL
LIN {X 0,Y 608.436,Z 110.317,A -85,B 0,C 180,E1 -490.327,E2 -490.327} C_VEL
LIN {X 0,Y 608.478,Z 110.313,A -85,B 0,C 180,E1 -493.31,E2 -493.31} C_VEL
LIN {X 0,Y 608.457,Z 110.315,A -85,B 0,C 180,E1 -496.13,E2 -496.13} C_VEL
LIN {X 0,Y 608.452,Z 110.313,A -85,B 0,C 180,E1 -498.823,E2 -498.823} C_VEL
LIN {X 0,Y 608.453,Z 110.318,A -85,B 0,C 180,E1 -501.762,E2 -501.762} C_VEL
LIN {X 0,Y 608.439,Z 110.317,A -85,B 0,C 180,E1 -503.956,E2 -503.956} C_VEL
LIN {X 0,Y 608.444,Z 110.314,A -85,B 0,C 180,E1 -506.328,E2 -506.328} C_VEL
LIN {X 0,Y 608.449,Z 110.315,A -85,B 0,C 180,E1 -508.732,E2 -508.732} C_VEL
LIN {X 0,Y 608.466,Z 110.318,A -85,B 0,C 180,E1 -511.382,E2 -511.382} C_VEL
LIN {X 0,Y 608.428,Z 110.316,A -85,B 0,C 180,E1 -513.964,E2 -513.964} C_VEL
LIN {X 0,Y 608.447,Z 110.321,A -85,B 0,C 180,E1 -516.876,E2 -516.876} C_VEL
LIN {X 0,Y 608.449,Z 110.318,A -85,B 0,C 180,E1 -519.327,E2 -519.327} C_VEL
LIN {X 0,Y 608.425,Z 110.316,A -85,B 0,C 180,E1 -521.827,E2 -521.827} C_VEL
LIN {X 0,Y 608.473,Z 110.316,A -85,B 0,C 180,E1 -524.594,E2 -524.594} C_VEL
LIN {X 0,Y 608.426,Z 110.318,A -85,B 0,C 180,E1 -527.322,E2 -527.322} C_VEL
LIN {X 0,Y 608.433,Z 110.316,A -85,B 0,C 180,E1 -529.35,E2 -529.35} C_VEL
LIN {X 0,Y 608.472,Z 110.312,A -85,B 0,C 180,E1 -532.033,E2 -532.033} C_VEL
LIN {X 0,Y 608.457,Z 110.32,A -85,B 0,C 180,E1 -534.698,E2 -534.698} C_VEL
LIN {X 0,Y 608.442,Z 110.314,A -85,B 0,C 180,E1 -537.352,E2 -537.352} C_VEL
LIN {X 0,Y 608.477,Z 110.313,A -85,B 0,C 180,E1 -540,E2 -540} C_VEL
LIN {X 0,Y 608.458,Z 110.317,A -85,B 0,C 180,E1 -542.648,E2 -542.648} C_VEL
LIN {X 0,Y 608.429,Z 110.315,A -85,B 0,C 180,E1 -545.302,E2 -545.302} C_VEL
LIN {X 0,Y 608.477,Z 110.316,A -85,B 0,C 180,E1 -547.967,E2 -547.967} C_VEL
LIN {X 0,Y 608.437,Z 110.315,A -85,B 0,C 180,E1 -549.435,E2 -549.435} C_VEL
LIN {X 0,Y 607.779,Z 110.405,A -85,B 0,C 180,E1 -549.988,E2 -549.988} C_VEL
LIN {X 0,Y 604.943,Z 110.762,A -85,B 0,C 180,E1 -550.884,E2 -550.884} C_VEL
LIN {X 0,Y 602.532,Z 111.062,A -85,B 0,C 180,E1 -551.606,E2 -551.606} C_VEL
LIN {X 0,Y 601.48,Z 111.19,A -85,B 0,C 180,E1 -552.162,E2 -552.162} C_VEL
LIN {X 0,Y 601.386,Z 111.198,A -85,B 0,C 180,E1 -552.351,E2 -552.351} C_VEL
LIN {X 0,Y 601.384,Z 111.193,A -85,B 0,C 180,E1 -554.898,E2 -554.898} C_VEL
LIN {X 0,Y 601.377,Z 111.194,A -85,B 0,C 180,E1 -556.988,E2 -556.988} C_VEL
LIN {X 0,Y 601.389,Z 111.203,A -85,B 0,C 180,E1 -559.81,E2 -559.81} C_VEL
LIN {X 0,Y 601.401,Z 111.191,A -85,B 0,C 180,E1 -562.684,E2 -562.684} C_VEL
LIN {X 0,Y 601.436,Z 111.196,A -85,B 0,C 180,E1 -565.617,E2 -565.617} C_VEL
LIN {X 0,Y 601.363,Z 111.202,A -85,B 0,C 180,E1 -567.87,E2 -567.87} C_VEL
LIN {X 0,Y 601.375,Z 111.196,A -85,B 0,C 180,E1 -570.167,E2 -570.167} C_VEL
LIN {X 0,Y 601.39,Z 111.193,A -85,B 0,C 180,E1 -572.71,E2 -572.71} C_VEL
LIN {X 0,Y 601.372,Z 111.2,A -85,B 0,C 180,E1 -575.108,E2 -575.108} C_VEL
LIN {X 0,Y 601.431,Z 111.196,A -85,B 0,C 180,E1 -577.419,E2 -577.419} C_VEL
LIN {X 0,Y 601.376,Z 111.195,A -85,B 0,C 180,E1 -579.998,E2 -579.998} C_VEL
LIN {X 0,Y 601.369,Z 111.197,A -85,B 0,C 180,E1 -582.674,E2 -582.674} C_VEL
LIN {X 0,Y 601.401,Z 111.196,A -85,B 0,C 180,E1 -585.479,E2 -585.479} C_VEL
LIN {X 0,Y 601.401,Z 111.193,A -85,B 0,C 180,E1 -588.409,E2 -588.409} C_VEL
LIN {X 0,Y 601.396,Z 111.201,A -85,B 0,C 180,E1 -590.872,E2 -590.872} C_VEL
LIN {X 0,Y 601.378,Z 111.196,A -85,B 0,C 180,E1 -593.415,E2 -593.415} C_VEL
LIN {X 0,Y 601.382,Z 111.194,A -85,B 0,C 180,E1 -596.072,E2 -596.072} C_VEL
LIN {X 0,Y 601.389,Z 111.2,A -85,B 0,C 180,E1 -598.55,E2 -598.55} C_VEL
LIN {X 0,Y 601.378,Z 111.195,A -85,B 0,C 180,E1 -601.37,E2 -601.37} C_VEL
LIN {X 0,Y 601.362,Z 111.196,A -85,B 0,C 180,E1 -603.634,E2 -603.634} C_VEL
LIN {X 0,Y 601.386,Z 111.195,A -85,B 0,C 180,E1 -605.857,E2 -605.857} C_VEL
LIN {X 0,Y 601.374,Z 111.259,A -85,B 0,C 180,E1 -607.44,E2 -607.44} C_VEL
LIN {X 0,Y 601.669,Z 118.429,A -85,B 0,C 180,E1 -608.411,E2 -608.411} C_VEL
LIN {X 0,Y 601.578,Z 139.942,A -85,B 0,C 180,E1 -611.25,E2 -611.25} C_VEL
LIN {X 0,Y 601.577,Z 140.859,A -85,B 0,C 180,E1 -611.37,E2 -611.37} C_VEL
LIN {X 0,Y 602.01,Z 144.875,A -85,B 0,C 180,E1 -611.443,E2 -611.443} C_VEL
LIN {X 0,Y 601.869,Z 306.209,A -85,B 0,C 180,E1 -613.436,E2 -613.436} C_VEL
LIN {X 0,Y 601.851,Z 321.659,A -85,B 0,C 180,E1 -613.768,E2 -613.768} C_VEL
LIN {X 0,Y 601.767,Z 337.007,A -85,B 0,C 180,E1 -614.244,E2 -614.244} C_VEL
LIN {X 0,Y 601.706,Z 351.684,A -85,B 0,C 180,E1 -614.85,E2 -614.85} C_VEL
LIN {X 0,Y 601.657,Z 364.983,A -85,B 0,C 180,E1 -615.541,E2 -615.541} C_VEL
LIN {X 0,Y 601.604,Z 377.802,A -85,B 0,C 180,E1 -616.352,E2 -616.352} C_VEL
LIN {X 0,Y 601.541,Z 389.789,A -85,B 0,C 180,E1 -617.26,E2 -617.26} C_VEL
LIN {X 0,Y 601.489,Z 400.28,A -85,B 0,C 180,E1 -618.201,E2 -618.201} C_VEL
LIN {X 0,Y 601.43,Z 409.996,A -85,B 0,C 180,E1 -619.224,E2 -619.224} C_VEL
LIN {X 0,Y 601.428,Z 419.526,A -85,B 0,C 180,E1 -620.415,E2 -620.415} C_VEL
LIN {X 0,Y 601.378,Z 427.46,A -85,B 0,C 180,E1 -621.6,E2 -621.6} C_VEL
LIN {X 0,Y 601.368,Z 434.872,A -85,B 0,C 180,E1 -622.951,E2 -622.951} C_VEL
LIN {X 0,Y 601.373,Z 440.759,A -85,B 0,C 180,E1 -624.299,E2 -624.299} C_VEL
LIN {X 0,Y 601.327,Z 444.241,A -85,B 0,C 180,E1 -625.307,E2 -625.307} C_VEL
LIN {X 0,Y 601.336,Z 447.79,A -85,B 0,C 180,E1 -626.65,E2 -626.65} C_VEL
LIN {X 0,Y 601.343,Z 450.139,A -85,B 0,C 180,E1 -627.991,E2 -627.991} C_VEL
LIN {X 0,Y 601.334,Z 451.337,A -85,B 0,C 180,E1 -629.33,E2 -629.33} C_VEL
LIN {X 0,Y 601.335,Z 451.361,A -85,B 0,C 180,E1 -630.67,E2 -630.67} C_VEL
LIN {X 0,Y 601.343,Z 450.245,A -85,B 0,C 180,E1 -632.009,E2 -632.009} C_VEL
LIN {X 0,Y 601.339,Z 447.983,A -85,B 0,C 180,E1 -633.35,E2 -633.35} C_VEL
LIN {X 0,Y 601.328,Z 444.525,A -85,B 0,C 180,E1 -634.693,E2 -634.693} C_VEL
LIN {X 0,Y 601.358,Z 439.797,A -85,B 0,C 180,E1 -636.038,E2 -636.038} C_VEL
LIN {X 0,Y 601.366,Z 433.666,A -85,B 0,C 180,E1 -637.386,E2 -637.386} C_VEL
LIN {X 0,Y 601.389,Z 425.95,A -85,B 0,C 180,E1 -638.738,E2 -638.738} C_VEL
LIN {X 0,Y 601.428,Z 417.706,A -85,B 0,C 180,E1 -639.925,E2 -639.925} C_VEL
LIN {X 0,Y 601.443,Z 407.365,A -85,B 0,C 180,E1 -641.164,E2 -641.164} C_VEL
LIN {X 0,Y 601.501,Z 395.784,A -85,B 0,C 180,E1 -642.312,E2 -642.312} C_VEL
LIN {X 0,Y 601.557,Z 384.462,A -85,B 0,C 180,E1 -643.255,E2 -643.255} C_VEL
LIN {X 0,Y 601.624,Z 371.312,A -85,B 0,C 180,E1 -644.168,E2 -644.168} C_VEL
LIN {X 0,Y 601.655,Z 358.756,A -85,B 0,C 180,E1 -644.891,E2 -644.891} C_VEL
LIN {X 0,Y 601.741,Z 343.831,A -85,B 0,C 180,E1 -645.583,E2 -645.583} C_VEL
LIN {X 0,Y 601.817,Z 329.341,A -85,B 0,C 180,E1 -646.102,E2 -646.102} C_VEL
LIN {X 0,Y 601.863,Z 314.206,A -85,B 0,C 180,E1 -646.5,E2 -646.5} C_VEL
LIN {X 0,Y 601.869,Z 298.831,A -85,B 0,C 180,E1 -646.762,E2 -646.762} C_VEL
LIN {X 0,Y 601.936,Z 142.708,A -85,B 0,C 180,E1 -648.676,E2 -648.676} C_VEL
LIN {X 0,Y 601.551,Z 140.82,A -85,B 0,C 180,E1 -648.726,E2 -648.726} C_VEL
LIN {X 0,Y 601.65,Z 120.454,A -85,B 0,C 180,E1 -651.41,E2 -651.41} C_VEL
LIN {X 0,Y 601.421,Z 111.572,A -85,B 0,C 180,E1 -652.606,E2 -652.606} C_VEL
LIN {X 0,Y 601.363,Z 111.2,A -85,B 0,C 180,E1 -652.685,E2 -652.685} C_VEL
LIN {X 0,Y 601.373,Z 111.197,A -85,B 0,C 180,E1 -654.88,E2 -654.88} C_VEL
LIN {X 0,Y 601.395,Z 111.201,A -85,B 0,C 180,E1 -657.358,E2 -657.358} C_VEL
LIN {X 0,Y 601.37,Z 111.196,A -85,B 0,C 180,E1 -660.167,E2 -660.167} C_VEL
LIN {X 0,Y 601.381,Z 111.196,A -85,B 0,C 180,E1 -662.709,E2 -662.709} C_VEL
LIN {X 0,Y 601.362,Z 111.204,A -85,B 0,C 180,E1 -665.107,E2 -665.107} C_VEL
LIN {X 0,Y 601.393,Z 111.198,A -85,B 0,C 180,E1 -667.422,E2 -667.422} C_VEL
LIN {X 0,Y 601.355,Z 111.197,A -85,B 0,C 180,E1 -670,E2 -670} C_VEL
LIN {X 0,Y 601.364,Z 111.2,A -85,B 0,C 180,E1 -672.675,E2 -672.675} C_VEL
LIN {X 0,Y 601.373,Z 111.197,A -85,B 0,C 180,E1 -675.477,E2 -675.477} C_VEL
LIN {X 0,Y 601.375,Z 111.195,A -85,B 0,C 180,E1 -678.231,E2 -678.231} C_VEL
LIN {X 0,Y 601.394,Z 111.2,A -85,B 0,C 180,E1 -680.872,E2 -680.872} C_VEL
LIN {X 0,Y 601.379,Z 111.194,A -85,B 0,C 180,E1 -683.415,E2 -683.415} C_VEL
LIN {X 0,Y 601.399,Z 111.194,A -85,B 0,C 180,E1 -686.07,E2 -686.07} C_VEL
LIN {X 0,Y 601.388,Z 111.195,A -85,B 0,C 180,E1 -689.056,E2 -689.056} C_VEL
LIN {X 0,Y 601.386,Z 111.193,A -85,B 0,C 180,E1 -691.371,E2 -691.371} C_VEL
LIN {X 0,Y 601.402,Z 111.197,A -85,B 0,C 180,E1 -694.136,E2 -694.136} C_VEL
LIN {X 0,Y 601.378,Z 111.2,A -85,B 0,C 180,E1 -696.588,E2 -696.588} C_VEL
LIN {X 0,Y 601.394,Z 111.193,A -85,B 0,C 180,E1 -699.477,E2 -699.477} C_VEL
LIN {X 0,Y 601.373,Z 111.196,A -85,B 0,C 180,E1 -701.607,E2 -701.607} C_VEL
LIN {X 0,Y 601.393,Z 111.197,A -85,B 0,C 180,E1 -704.408,E2 -704.408} C_VEL
LIN {X 0,Y 601.401,Z 111.194,A -85,B 0,C 180,E1 -706.484,E2 -706.484} C_VEL
LIN {X 0,Y 601.369,Z 111.196,A -85,B 0,C 180,E1 -709.223,E2 -709.223} C_VEL
LIN {X 0,Y 601.436,Z 111.196,A -85,B 0,C 180,E1 -711.939,E2 -711.939} C_VEL
LIN {X 0,Y 601.399,Z 111.191,A -85,B 0,C 180,E1 -714.636,E2 -714.636} C_VEL
LIN {X 0,Y 601.415,Z 111.193,A -85,B 0,C 180,E1 -717.321,E2 -717.321} C_VEL
LIN {X 0,Y 601.446,Z 111.19,A -85,B 0,C 180,E1 -720,E2 -720} C_VEL
LIN {X 0,Y 601.409,Z 111.19,A -85,B 0,C 180,E1 -722.679,E2 -722.679} C_VEL
LIN {X 0,Y 601.419,Z 111.197,A -85,B 0,C 180,E1 -725.364,E2 -725.364} C_VEL
LIN {X 0,Y 601.433,Z 111.188,A -85,B 0,C 180,E1 -728.061,E2 -728.061} C_VEL
LIN {X 0,Y 601.409,Z 111.195,A -85,B 0,C 180,E1 -731.002,E2 -731.002} C_VEL
LIN {X 0,Y 601.4,Z 111.191,A -85,B 0,C 180,E1 -734.082,E2 -734.082} C_VEL
LIN {X 0,Y 601.409,Z 111.198,A -85,B 0,C 180,E1 -736.986,E2 -736.986} C_VEL
LIN {X 0,Y 601.396,Z 111.193,A -85,B 0,C 180,E1 -739.81,E2 -739.81} C_VEL
LIN {X 0,Y 601.405,Z 111.196,A -85,B 0,C 180,E1 -742.683,E2 -742.683} C_VEL
LIN {X 0,Y 601.428,Z 111.188,A -85,B 0,C 180,E1 -745.618,E2 -745.618} C_VEL
LIN {X 0,Y 601.392,Z 111.192,A -85,B 0,C 180,E1 -747.869,E2 -747.869} C_VEL
LIN {X 0,Y 601.401,Z 111.193,A -85,B 0,C 180,E1 -750.165,E2 -750.165} C_VEL
LIN {X 0,Y 601.417,Z 111.199,A -85,B 0,C 180,E1 -752.714,E2 -752.714} C_VEL
LIN {X 0,Y 601.396,Z 111.195,A -85,B 0,C 180,E1 -755.112,E2 -755.112} C_VEL
LIN {X 0,Y 601.435,Z 111.187,A -85,B 0,C 180,E1 -757.419,E2 -757.419} C_VEL
LIN {X 0,Y 601.401,Z 111.194,A -85,B 0,C 180,E1 -759.996,E2 -759.996} C_VEL
LIN {X 0,Y 601.415,Z 111.195,A -85,B 0,C 180,E1 -762.67,E2 -762.67} C_VEL
LIN {X 0,Y 601.4,Z 111.192,A -85,B 0,C 180,E1 -765.479,E2 -765.479} C_VEL
LIN {X 0,Y 601.423,Z 111.195,A -85,B 0,C 180,E1 -768.407,E2 -768.407} C_VEL
LIN {X 0,Y 601.432,Z 111.188,A -85,B 0,C 180,E1 -770.875,E2 -770.875} C_VEL
LIN {X 0,Y 601.399,Z 111.193,A -85,B 0,C 180,E1 -773.416,E2 -773.416} C_VEL
LIN {X 0,Y 601.432,Z 111.197,A -85,B 0,C 180,E1 -776.064,E2 -776.064} C_VEL
LIN {X 0,Y 601.413,Z 111.19,A -85,B 0,C 180,E1 -779.057,E2 -779.057} C_VEL
LIN {X 0,Y 601.421,Z 111.192,A -85,B 0,C 180,E1 -781.372,E2 -781.372} C_VEL
LIN {X 0,Y 601.398,Z 111.2,A -85,B 0,C 180,E1 -783.636,E2 -783.636} C_VEL
LIN {X 0,Y 601.431,Z 111.226,A -85,B 0,C 180,E1 -784.521,E2 -784.521} C_VEL
LIN {X 0,Y 601.867,Z 114.738,A -85,B 0,C 180,E1 -784.957,E2 -784.957} C_VEL
LIN {X 0,Y 601.768,Z 138.192,A -85,B 0,C 180,E1 -787.698,E2 -787.698} C_VEL
LIN {X 0,Y 601.67,Z 163.118,A -85,B 0,C 180,E1 -790.555,E2 -790.555} C_VEL
LIN {X 0,Y 601.629,Z 169.87,A -85,B 0,C 180,E1 -791.319,E2 -791.319} C_VEL
LIN {X 0,Y 602.027,Z 174.028,A -85,B 0,C 180,E1 -791.388,E2 -791.388} C_VEL
LIN {X 0,Y 601.887,Z 335.267,A -85,B 0,C 180,E1 -793.377,E2 -793.377} C_VEL
LIN {X 0,Y 601.86,Z 350.883,A -85,B 0,C 180,E1 -793.704,E2 -793.704} C_VEL
LIN {X 0,Y 601.797,Z 365.789,A -85,B 0,C 180,E1 -794.158,E2 -794.158} C_VEL
LIN {X 0,Y 601.723,Z 380.758,A -85,B 0,C 180,E1 -794.764,E2 -794.764} C_VEL
LIN {X 0,Y 601.658,Z 394.232,A -85,B 0,C 180,E1 -795.455,E2 -795.455} C_VEL
LIN {X 0,Y 601.617,Z 407.449,A -85,B 0,C 180,E1 -796.283,E2 -796.283} C_VEL
LIN {X 0,Y 601.531,Z 419.284,A -85,B 0,C 180,E1 -797.174,E2 -797.174} C_VEL
LIN {X 0,Y 601.488,Z 430.747,A -85,B 0,C 180,E1 -798.201,E2 -798.201} C_VEL
LIN {X 0,Y 601.43,Z 440.388,A -85,B 0,C 180,E1 -799.224,E2 -799.224} C_VEL
LIN {X 0,Y 601.428,Z 449.854,A -85,B 0,C 180,E1 -800.414,E2 -800.414} C_VEL
LIN {X 0,Y 601.369,Z 457.73,A -85,B 0,C 180,E1 -801.6,E2 -801.6} C_VEL
LIN {X 0,Y 601.367,Z 465.087,A -85,B 0,C 180,E1 -802.951,E2 -802.951} C_VEL
LIN {X 0,Y 601.373,Z 470.924,A -85,B 0,C 180,E1 -804.299,E2 -804.299} C_VEL
LIN {X 0,Y 601.33,Z 474.383,A -85,B 0,C 180,E1 -805.307,E2 -805.307} C_VEL
LIN {X 0,Y 601.337,Z 477.886,A -85,B 0,C 180,E1 -806.65,E2 -806.65} C_VEL
LIN {X 0,Y 601.343,Z 480.192,A -85,B 0,C 180,E1 -807.991,E2 -807.991} C_VEL
LIN {X 0,Y 601.335,Z 481.35,A -85,B 0,C 180,E1 -809.33,E2 -809.33} C_VEL
LIN {X 0,Y 601.335,Z 481.35,A -85,B 0,C 180,E1 -810.67,E2 -810.67} C_VEL
LIN {X 0,Y 601.343,Z 480.192,A -85,B 0,C 180,E1 -812.009,E2 -812.009} C_VEL
LIN {X 0,Y 601.337,Z 477.886,A -85,B 0,C 180,E1 -813.35,E2 -813.35} C_VEL
LIN {X 0,Y 601.33,Z 474.383,A -85,B 0,C 180,E1 -814.693,E2 -814.693} C_VEL
LIN {X 0,Y 601.357,Z 469.608,A -85,B 0,C 180,E1 -816.038,E2 -816.038} C_VEL
LIN {X 0,Y 601.365,Z 463.425,A -85,B 0,C 180,E1 -817.386,E2 -817.386} C_VEL
LIN {X 0,Y 601.388,Z 455.653,A -85,B 0,C 180,E1 -818.738,E2 -818.738} C_VEL
LIN {X 0,Y 601.427,Z 447.37,A -85,B 0,C 180,E1 -819.925,E2 -819.925} C_VEL
LIN {X 0,Y 601.46,Z 436.932,A -85,B 0,C 180,E1 -821.165,E2 -821.165} C_VEL
LIN {X 0,Y 601.514,Z 427.191,A -85,B 0,C 180,E1 -822.141,E2 -822.141} C_VEL
LIN {X 0,Y 601.57,Z 415.015,A -85,B 0,C 180,E1 -823.168,E2 -823.168} C_VEL
LIN {X 0,Y 601.606,Z 403.075,A -85,B 0,C 180,E1 -824.012,E2 -824.012} C_VEL
LIN {X 0,Y 601.65,Z 389.524,A -85,B 0,C 180,E1 -824.805,E2 -824.805} C_VEL
LIN {X 0,Y 601.771,Z 374.84,A -85,B 0,C 180,E1 -825.495,E2 -825.495} C_VEL
LIN {X 0,Y 601.793,Z 360.615,A -85,B 0,C 180,E1 -826.016,E2 -826.016} C_VEL
LIN {X 0,Y 601.856,Z 345.696,A -85,B 0,C 180,E1 -826.42,E2 -826.42} C_VEL
LIN {X 0,Y 601.868,Z 330.718,A -85,B 0,C 180,E1 -826.69,E2 -826.69} C_VEL
LIN {X 0,Y 601.905,Z 171.467,A -85,B 0,C 180,E1 -828.647,E2 -828.647} C_VEL
LIN {X 0,Y 601.628,Z 169.747,A -85,B 0,C 180,E1 -828.695,E2 -828.695} C_VEL
LIN {X 0,Y 601.75,Z 144.391,A -85,B 0,C 180,E1 -831.586,E2 -831.586} C_VEL
LIN {X 0,Y 601.868,Z 120.326,A -85,B 0,C 180,E1 -834.383,E2 -834.383} C_VEL
LIN {X 0,Y 601.853,Z 113.177,A -85,B 0,C 180,E1 -835.228,E2 -835.228} C_VEL
LIN {X 0,Y 601.437,Z 111.192,A -85,B 0,C 180,E1 -835.501,E2 -835.501} C_VEL
LIN {X 0,Y 601.402,Z 111.197,A -85,B 0,C 180,E1 -837.868,E2 -837.868} C_VEL
LIN {X 0,Y 601.429,Z 111.197,A -85,B 0,C 180,E1 -840.164,E2 -840.164} C_VEL
LIN {X 0,Y 601.413,Z 111.19,A -85,B 0,C 180,E1 -842.714,E2 -842.714} C_VEL
LIN {X 0,Y 601.389,Z 111.193,A -85,B 0,C 180,E1 -845.111,E2 -845.111} C_VEL
LIN {X 0,Y 601.436,Z 111.19,A -85,B 0,C 180,E1 -847.419,E2 -847.419} C_VEL
LIN {X 0,Y 601.413,Z 111.197,A -85,B 0,C 180,E1 -849.995,E2 -849.995} C_VEL
LIN {X 0,Y 601.407,Z 111.19,A -85,B 0,C 180,E1 -852.671,E2 -852.671} C_VEL
LIN {X 0,Y 601.428,Z 111.195,A -85,B 0,C 180,E1 -855.482,E2 -855.482} C_VEL
LIN {X 0,Y 601.417,Z 111.189,A -85,B 0,C 180,E1 -858.408,E2 -858.408} C_VEL
LIN {X 0,Y 601.414,Z 111.191,A -85,B 0,C 180,E1 -860.874,E2 -860.874} C_VEL
LIN {X 0,Y 601.405,Z 111.201,A -85,B 0,C 180,E1 -863.417,E2 -863.417} C_VEL
LIN {X 0,Y 601.418,Z 111.19,A -85,B 0,C 180,E1 -866.067,E2 -866.067} C_VEL
LIN {X 0,Y 601.419,Z 111.189,A -85,B 0,C 180,E1 -868.546,E2 -868.546} C_VEL
LIN {X 0,Y 601.427,Z 111.195,A -85,B 0,C 180,E1 -871.373,E2 -871.373} C_VEL
LIN {X 0,Y 601.393,Z 111.195,A -85,B 0,C 180,E1 -873.636,E2 -873.636} C_VEL
LIN {X 0,Y 601.41,Z 111.19,A -85,B 0,C 180,E1 -875.858,E2 -875.858} C_VEL
LIN {X 0,Y 601.404,Z 111.197,A -85,B 0,C 180,E1 -878.761,E2 -878.761} C_VEL
LIN {X 0,Y 601.386,Z 111.194,A -85,B 0,C 180,E1 -881.607,E2 -881.607} C_VEL
LIN {X 0,Y 601.411,Z 111.193,A -85,B 0,C 180,E1 -884.409,E2 -884.409} C_VEL
LIN {X 0,Y 601.384,Z 111.197,A -85,B 0,C 180,E1 -887.171,E2 -887.171} C_VEL
LIN {X 0,Y 601.393,Z 111.195,A -85,B 0,C 180,E1 -889.224,E2 -889.224} C_VEL
LIN {X 0,Y 601.433,Z 111.188,A -85,B 0,C 180,E1 -891.939,E2 -891.939} C_VEL
LIN {X 0,Y 601.423,Z 111.197,A -85,B 0,C 180,E1 -894.636,E2 -894.636} C_VEL
LIN {X 0,Y 601.412,Z 111.19,A -85,B 0,C 180,E1 -897.321,E2 -897.321} C_VEL
LIN {X 0,Y 601.446,Z 111.189,A -85,B 0,C 180,E1 -900,E2 -900} C_VEL
LIN {X 0,Y 601.423,Z 111.193,A -85,B 0,C 180,E1 -902.679,E2 -902.679} C_VEL
LIN {X 0,Y 601.401,Z 111.191,A -85,B 0,C 180,E1 -905.364,E2 -905.364} C_VEL
LIN {X 0,Y 601.437,Z 111.195,A -85,B 0,C 180,E1 -908.061,E2 -908.061} C_VEL
LIN {X 0,Y 601.389,Z 111.193,A -85,B 0,C 180,E1 -910.993,E2 -910.993} C_VEL
LIN {X 0,Y 601.386,Z 111.198,A -85,B 0,C 180,E1 -912.351,E2 -912.351} C_VEL
LIN {X 0,Y 600.697,Z 111.281,A -85,B 0,C 180,E1 -912.91,E2 -912.91} C_VEL
LIN {X 0,Y 597.84,Z 111.641,A -85,B 0,C 180,E1 -913.818,E2 -913.818} C_VEL
LIN {X 0,Y 595.442,Z 111.936,A -85,B 0,C 180,E1 -914.549,E2 -914.549} C_VEL
LIN {X 0,Y 594.415,Z 112.062,A -85,B 0,C 180,E1 -915.112,E2 -915.112} C_VEL
LIN {X 0,Y 594.332,Z 112.073,A -85,B 0,C 180,E1 -915.303,E2 -915.303} C_VEL
LIN {X 0,Y 594.333,Z 112.082,A -85,B 0,C 180,E1 -917.906,E2 -917.906} C_VEL
LIN {X 0,Y 594.376,Z 112.066,A -85,B 0,C 180,E1 -920.777,E2 -920.777} C_VEL
LIN {X 0,Y 594.352,Z 112.079,A -85,B 0,C 180,E1 -923.706,E2 -923.706} C_VEL
LIN {X 0,Y 594.357,Z 112.071,A -85,B 0,C 180,E1 -926.016,E2 -926.016} C_VEL
LIN {X 0,Y 594.369,Z 112.069,A -85,B 0,C 180,E1 -928.999,E2 -928.999} C_VEL
LIN {X 0,Y 594.368,Z 112.075,A -85,B 0,C 180,E1 -931.641,E2 -931.641} C_VEL
LIN {X 0,Y 594.358,Z 112.069,A -85,B 0,C 180,E1 -934.135,E2 -934.135} C_VEL
LIN {X 0,Y 594.377,Z 112.072,A -85,B 0,C 180,E1 -937.087,E2 -937.087} C_VEL
LIN {X 0,Y 594.337,Z 112.074,A -85,B 0,C 180,E1 -939.769,E2 -939.769} C_VEL
LIN {X 0,Y 594.329,Z 112.072,A -85,B 0,C 180,E1 -942.379,E2 -942.379} C_VEL
LIN {X 0,Y 594.339,Z 112.08,A -85,B 0,C 180,E1 -945.194,E2 -945.194} C_VEL
LIN {X 0,Y 594.353,Z 112.069,A -85,B 0,C 180,E1 -948.155,E2 -948.155} C_VEL
LIN {X 0,Y 594.357,Z 112.075,A -85,B 0,C 180,E1 -951.193,E2 -951.193} C_VEL
LIN {X 0,Y 594.311,Z 112.075,A -85,B 0,C 180,E1 -953.752,E2 -953.752} C_VEL
LIN {X 0,Y 594.334,Z 112.074,A -85,B 0,C 180,E1 -956.236,E2 -956.236} C_VEL
LIN {X 0,Y 594.34,Z 112.08,A -85,B 0,C 180,E1 -958.648,E2 -958.648} C_VEL
LIN {X 0,Y 594.337,Z 112.076,A -85,B 0,C 180,E1 -961.051,E2 -961.051} C_VEL
LIN {X 0,Y 594.348,Z 112.071,A -85,B 0,C 180,E1 -963.299,E2 -963.299} C_VEL
LIN {X 0,Y 594.332,Z 112.08,A -85,B 0,C 180,E1 -966.293,E2 -966.293} C_VEL
LIN {X 0,Y 594.324,Z 112.126,A -85,B 0,C 180,E1 -967.275,E2 -967.275} C_VEL
LIN {X 0,Y 594.74,Z 117.084,A -85,B 0,C 180,E1 -967.964,E2 -967.964} C_VEL
LIN {X 0,Y 594.669,Z 137.326,A -85,B 0,C 180,E1 -970.676,E2 -970.676} C_VEL
LIN {X 0,Y 594.619,Z 140.921,A -85,B 0,C 180,E1 -971.151,E2 -971.151} C_VEL
LIN {X 0,Y 595.288,Z 145.088,A -85,B 0,C 180,E1 -971.228,E2 -971.228} C_VEL
LIN {X 0,Y 595.063,Z 306.553,A -85,B 0,C 180,E1 -973.247,E2 -973.247} C_VEL
LIN {X 0,Y 595.028,Z 322.457,A -85,B 0,C 180,E1 -973.599,E2 -973.599} C_VEL
LIN {X 0,Y 594.924,Z 337.021,A -85,B 0,C 180,E1 -974.058,E2 -974.058} C_VEL
LIN {X 0,Y 594.821,Z 351.694,A -85,B 0,C 180,E1 -974.671,E2 -974.671} C_VEL
LIN {X 0,Y 594.742,Z 364.997,A -85,B 0,C 180,E1 -975.369,E2 -975.369} C_VEL
LIN {X 0,Y 594.67,Z 377.99,A -85,B 0,C 180,E1 -976.201,E2 -976.201} C_VEL
LIN {X 0,Y 594.552,Z 390.858,A -85,B 0,C 180,E1 -977.195,E2 -977.195} C_VEL
LIN {X 0,Y 594.468,Z 402.062,A -85,B 0,C 180,E1 -978.233,E2 -978.233} C_VEL
LIN {X 0,Y 594.412,Z 412.946,A -85,B 0,C 180,E1 -979.44,E2 -979.44} C_VEL
LIN {X 0,Y 594.357,Z 421.99,A -85,B 0,C 180,E1 -980.643,E2 -980.643} C_VEL
LIN {X 0,Y 594.324,Z 429.485,A -85,B 0,C 180,E1 -981.842,E2 -981.842} C_VEL
LIN {X 0,Y 594.277,Z 436.49,A -85,B 0,C 180,E1 -983.208,E2 -983.208} C_VEL
LIN {X 0,Y 594.273,Z 441.999,A -85,B 0,C 180,E1 -984.571,E2 -984.571} C_VEL
LIN {X 0,Y 594.253,Z 446.171,A -85,B 0,C 180,E1 -985.931,E2 -985.931} C_VEL
LIN {X 0,Y 594.221,Z 449.112,A -85,B 0,C 180,E1 -987.288,E2 -987.288} C_VEL
LIN {X 0,Y 594.243,Z 450.88,A -85,B 0,C 180,E1 -988.645,E2 -988.645} C_VEL
LIN {X 0,Y 594.234,Z 451.496,A -85,B 0,C 180,E1 -990,E2 -990} C_VEL
LIN {X 0,Y 594.245,Z 450.944,A -85,B 0,C 180,E1 -991.355,E2 -991.355} C_VEL
LIN {X 0,Y 594.224,Z 449.26,A -85,B 0,C 180,E1 -992.712,E2 -992.712} C_VEL
LIN {X 0,Y 594.253,Z 446.406,A -85,B 0,C 180,E1 -994.069,E2 -994.069} C_VEL
LIN {X 0,Y 594.273,Z 442.325,A -85,B 0,C 180,E1 -995.429,E2 -995.429} C_VEL
LIN {X 0,Y 594.277,Z 436.915,A -85,B 0,C 180,E1 -996.792,E2 -996.792} C_VEL
LIN {X 0,Y 594.323,Z 430.016,A -85,B 0,C 180,E1 -998.158,E2 -998.158} C_VEL
LIN {X 0,Y 594.339,Z 421.413,A -85,B 0,C 180,E1 -999.529,E2 -999.529} C_VEL
LIN {X 0,Y 594.401,Z 412.263,A -85,B 0,C 180,E1 -1000.733,E2 -1000.733} C_VEL
LIN {X 0,Y 594.466,Z 401.209,A -85,B 0,C 180,E1 -1001.94,E2 -1001.94} C_VEL
LIN {X 0,Y 594.56,Z 389.834,A -85,B 0,C 180,E1 -1002.979,E2 -1002.979} C_VEL
LIN {X 0,Y 594.66,Z 377.451,A -85,B 0,C 180,E1 -1003.925,E2 -1003.925} C_VEL
LIN {X 0,Y 594.722,Z 365.041,A -85,B 0,C 180,E1 -1004.719,E2 -1004.719} C_VEL
LIN {X 0,Y 594.828,Z 351.742,A -85,B 0,C 180,E1 -1005.417,E2 -1005.417} C_VEL
LIN {X 0,Y 594.921,Z 337.068,A -85,B 0,C 180,E1 -1006.03,E2 -1006.03} C_VEL
LIN {X 0,Y 595.027,Z 321.224,A -85,B 0,C 180,E1 -1006.525,E2 -1006.525} C_VEL
LIN {X 0,Y 595.084,Z 305.676,A -85,B 0,C 180,E1 -1006.858,E2 -1006.858} C_VEL
LIN {X 0,Y 595.226,Z 143.986,A -85,B 0,C 180,E1 -1008.878,E2 -1008.878} C_VEL
LIN {X 0,Y 594.626,Z 140.92,A -85,B 0,C 180,E1 -1008.939,E2 -1008.939} C_VEL
LIN {X 0,Y 594.761,Z 120.45,A -85,B 0,C 180,E1 -1011.67,E2 -1011.67} C_VEL
LIN {X 0,Y 594.704,Z 114.499,A -85,B 0,C 180,E1 -1012.478,E2 -1012.478} C_VEL
LIN {X 0,Y 594.312,Z 112.08,A -85,B 0,C 180,E1 -1012.849,E2 -1012.849} C_VEL
LIN {X 0,Y 594.331,Z 112.078,A -85,B 0,C 180,E1 -1015.195,E2 -1015.195} C_VEL
LIN {X 0,Y 594.344,Z 112.08,A -85,B 0,C 180,E1 -1017.518,E2 -1017.518} C_VEL
LIN {X 0,Y 594.345,Z 112.071,A -85,B 0,C 180,E1 -1020.321,E2 -1020.321} C_VEL
LIN {X 0,Y 594.338,Z 112.076,A -85,B 0,C 180,E1 -1022.953,E2 -1022.953} C_VEL
LIN {X 0,Y 594.299,Z 112.083,A -85,B 0,C 180,E1 -1025.413,E2 -1025.413} C_VEL
LIN {X 0,Y 594.299,Z 112.077,A -85,B 0,C 180,E1 -1027.948,E2 -1027.948} C_VEL
LIN {X 0,Y 594.355,Z 112.075,A -85,B 0,C 180,E1 -1030.819,E2 -1030.819} C_VEL
LIN {X 0,Y 594.341,Z 112.071,A -85,B 0,C 180,E1 -1033.837,E2 -1033.837} C_VEL
LIN {X 0,Y 594.34,Z 112.078,A -85,B 0,C 180,E1 -1036.698,E2 -1036.698} C_VEL
LIN {X 0,Y 594.339,Z 112.073,A -85,B 0,C 180,E1 -1039.43,E2 -1039.43} C_VEL
LIN {X 0,Y 594.375,Z 112.07,A -85,B 0,C 180,E1 -1042.394,E2 -1042.394} C_VEL
LIN {X 0,Y 594.353,Z 112.07,A -85,B 0,C 180,E1 -1045.418,E2 -1045.418} C_VEL
LIN {X 0,Y 594.336,Z 112.071,A -85,B 0,C 180,E1 -1047.851,E2 -1047.851} C_VEL
LIN {X 0,Y 594.337,Z 112.075,A -85,B 0,C 180,E1 -1050.221,E2 -1050.221} C_VEL
LIN {X 0,Y 594.354,Z 112.069,A -85,B 0,C 180,E1 -1053.299,E2 -1053.299} C_VEL
LIN {X 0,Y 594.337,Z 112.072,A -85,B 0,C 180,E1 -1055.578,E2 -1055.578} C_VEL
LIN {X 0,Y 594.349,Z 112.076,A -85,B 0,C 180,E1 -1058.496,E2 -1058.496} C_VEL
LIN {X 0,Y 594.348,Z 112.07,A -85,B 0,C 180,E1 -1061.381,E2 -1061.381} C_VEL
LIN {X 0,Y 594.343,Z 112.079,A -85,B 0,C 180,E1 -1064.218,E2 -1064.218} C_VEL
LIN {X 0,Y 594.371,Z 112.072,A -85,B 0,C 180,E1 -1066.321,E2 -1066.321} C_VEL
LIN {X 0,Y 594.347,Z 112.07,A -85,B 0,C 180,E1 -1069.094,E2 -1069.094} C_VEL
LIN {X 0,Y 594.379,Z 112.075,A -85,B 0,C 180,E1 -1071.843,E2 -1071.843} C_VEL
LIN {X 0,Y 594.37,Z 112.067,A -85,B 0,C 180,E1 -1074.572,E2 -1074.572} C_VEL
LIN {X 0,Y 594.382,Z 112.069,A -85,B 0,C 180,E1 -1077.289,E2 -1077.289} C_VEL
LIN {X 0,Y 594.415,Z 112.065,A -85,B 0,C 180,E1 -1080,E2 -1080} C_VEL
LIN {X 0,Y 594.379,Z 112.066,A -85,B 0,C 180,E1 -1082.711,E2 -1082.711} C_VEL
LIN {X 0,Y 594.385,Z 112.074,A -85,B 0,C 180,E1 -1085.428,E2 -1085.428} C_VEL
LIN {X 0,Y 594.377,Z 112.067,A -85,B 0,C 180,E1 -1088.157,E2 -1088.157} C_VEL
LIN {X 0,Y 594.374,Z 112.072,A -85,B 0,C 180,E1 -1091.064,E2 -1091.064} C_VEL
LIN {X 0,Y 594.373,Z 112.07,A -85,B 0,C 180,E1 -1093.679,E2 -1093.679} C_VEL
LIN {X 0,Y 594.359,Z 112.072,A -85,B 0,C 180,E1 -1096.707,E2 -1096.707} C_VEL
LIN {X 0,Y 594.364,Z 112.074,A -85,B 0,C 180,E1 -1099.334,E2 -1099.334} C_VEL
LIN {X 0,Y 594.359,Z 112.071,A -85,B 0,C 180,E1 -1101.503,E2 -1101.503} C_VEL
LIN {X 0,Y 594.346,Z 112.073,A -85,B 0,C 180,E1 -1104.448,E2 -1104.448} C_VEL
LIN {X 0,Y 594.382,Z 112.073,A -85,B 0,C 180,E1 -1106.7,E2 -1106.7} C_VEL
LIN {X 0,Y 594.381,Z 112.073,A -85,B 0,C 180,E1 -1108.998,E2 -1108.998} C_VEL
LIN {X 0,Y 594.375,Z 112.067,A -85,B 0,C 180,E1 -1111.642,E2 -1111.642} C_VEL
LIN {X 0,Y 594.38,Z 112.075,A -85,B 0,C 180,E1 -1114.58,E2 -1114.58} C_VEL
LIN {X 0,Y 594.387,Z 112.065,A -85,B 0,C 180,E1 -1117.608,E2 -1117.608} C_VEL
LIN {X 0,Y 594.365,Z 112.076,A -85,B 0,C 180,E1 -1120.567,E2 -1120.567} C_VEL
LIN {X 0,Y 594.368,Z 112.067,A -85,B 0,C 180,E1 -1123.299,E2 -1123.299} C_VEL
LIN {X 0,Y 594.362,Z 112.076,A -85,B 0,C 180,E1 -1126.161,E2 -1126.161} C_VEL
LIN {X 0,Y 594.381,Z 112.07,A -85,B 0,C 180,E1 -1128.536,E2 -1128.536} C_VEL
LIN {X 0,Y 594.379,Z 112.066,A -85,B 0,C 180,E1 -1131.296,E2 -1131.296} C_VEL
LIN {X 0,Y 594.351,Z 112.074,A -85,B 0,C 180,E1 -1133.755,E2 -1133.755} C_VEL
LIN {X 0,Y 594.379,Z 112.073,A -85,B 0,C 180,E1 -1136.239,E2 -1136.239} C_VEL
LIN {X 0,Y 594.37,Z 112.068,A -85,B 0,C 180,E1 -1138.65,E2 -1138.65} C_VEL
LIN {X 0,Y 594.382,Z 112.067,A -85,B 0,C 180,E1 -1141.042,E2 -1141.042} C_VEL
LIN {X 0,Y 594.386,Z 112.076,A -85,B 0,C 180,E1 -1143.977,E2 -1143.977} C_VEL
LIN {X 0,Y 594.4,Z 112.201,A -85,B 0,C 180,E1 -1144.316,E2 -1144.316} C_VEL
LIN {X 0,Y 595.072,Z 116.298,A -85,B 0,C 180,E1 -1144.838,E2 -1144.838} C_VEL
LIN {X 0,Y 594.911,Z 141.269,A -85,B 0,C 180,E1 -1147.788,E2 -1147.788} C_VEL
LIN {X 0,Y 594.751,Z 166.239,A -85,B 0,C 180,E1 -1150.678,E2 -1150.678} C_VEL
LIN {X 0,Y 594.701,Z 169.887,A -85,B 0,C 180,E1 -1151.095,E2 -1151.095} C_VEL
LIN {X 0,Y 595.313,Z 173.419,A -85,B 0,C 180,E1 -1151.163,E2 -1151.163} C_VEL
LIN {X 0,Y 595.081,Z 336.381,A -85,B 0,C 180,E1 -1153.199,E2 -1153.199} C_VEL
LIN {X 0,Y 595.014,Z 351.704,A -85,B 0,C 180,E1 -1153.532,E2 -1153.532} C_VEL
LIN {X 0,Y 594.944,Z 367.042,A -85,B 0,C 180,E1 -1154.015,E2 -1154.015} C_VEL
LIN {X 0,Y 594.863,Z 380.762,A -85,B 0,C 180,E1 -1154.584,E2 -1154.584} C_VEL
LIN {X 0,Y 594.732,Z 394.236,A -85,B 0,C 180,E1 -1155.282,E2 -1155.282} C_VEL
LIN {X 0,Y 594.681,Z 406.792,A -85,B 0,C 180,E1 -1156.075,E2 -1156.075} C_VEL
LIN {X 0,Y 594.56,Z 419.285,A -85,B 0,C 180,E1 -1157.021,E2 -1157.021} C_VEL
LIN {X 0,Y 594.465,Z 430.747,A -85,B 0,C 180,E1 -1158.06,E2 -1158.06} C_VEL
LIN {X 0,Y 594.388,Z 440.389,A -85,B 0,C 180,E1 -1159.095,E2 -1159.095} C_VEL
LIN {X 0,Y 594.366,Z 449.855,A -85,B 0,C 180,E1 -1160.299,E2 -1160.299} C_VEL
LIN {X 0,Y 594.312,Z 457.731,A -85,B 0,C 180,E1 -1161.499,E2 -1161.499} C_VEL
LIN {X 0,Y 594.292,Z 465.088,A -85,B 0,C 180,E1 -1162.867,E2 -1162.867} C_VEL
LIN {X 0,Y 594.299,Z 470.924,A -85,B 0,C 180,E1 -1164.231,E2 -1164.231} C_VEL
LIN {X 0,Y 594.232,Z 474.384,A -85,B 0,C 180,E1 -1165.251,E2 -1165.251} C_VEL
LIN {X 0,Y 594.257,Z 477.887,A -85,B 0,C 180,E1 -1166.61,E2 -1166.61} C_VEL
LIN {X 0,Y 594.241,Z 480.193,A -85,B 0,C 180,E1 -1167.967,E2 -1167.967} C_VEL
LIN {X 0,Y 594.235,Z 481.35,A -85,B 0,C 180,E1 -1169.322,E2 -1169.322} C_VEL
LIN {X 0,Y 594.235,Z 481.35,A -85,B 0,C 180,E1 -1170.678,E2 -1170.678} C_VEL
LIN {X 0,Y 594.241,Z 480.192,A -85,B 0,C 180,E1 -1172.033,E2 -1172.033} C_VEL
LIN {X 0,Y 594.257,Z 477.886,A -85,B 0,C 180,E1 -1173.39,E2 -1173.39} C_VEL
LIN {X 0,Y 594.232,Z 474.384,A -85,B 0,C 180,E1 -1174.749,E2 -1174.749} C_VEL
LIN {X 0,Y 594.279,Z 469.608,A -85,B 0,C 180,E1 -1176.11,E2 -1176.11} C_VEL
LIN {X 0,Y 594.287,Z 463.424,A -85,B 0,C 180,E1 -1177.475,E2 -1177.475} C_VEL
LIN {X 0,Y 594.331,Z 455.651,A -85,B 0,C 180,E1 -1178.843,E2 -1178.843} C_VEL
LIN {X 0,Y 594.387,Z 447.369,A -85,B 0,C 180,E1 -1180.044,E2 -1180.044} C_VEL
LIN {X 0,Y 594.433,Z 437.559,A -85,B 0,C 180,E1 -1181.231,E2 -1181.231} C_VEL
LIN {X 0,Y 594.53,Z 427.19,A -85,B 0,C 180,E1 -1182.285,E2 -1182.285} C_VEL
LIN {X 0,Y 594.581,Z 415.017,A -85,B 0,C 180,E1 -1183.326,E2 -1183.326} C_VEL
LIN {X 0,Y 594.694,Z 403.072,A -85,B 0,C 180,E1 -1184.178,E2 -1184.178} C_VEL
LIN {X 0,Y 594.751,Z 389.521,A -85,B 0,C 180,E1 -1184.981,E2 -1184.981} C_VEL
LIN {X 0,Y 594.913,Z 374.836,A -85,B 0,C 180,E1 -1185.678,E2 -1185.678} C_VEL
LIN {X 0,Y 594.972,Z 360.615,A -85,B 0,C 180,E1 -1186.205,E2 -1186.205} C_VEL
LIN {X 0,Y 595.046,Z 346.12,A -85,B 0,C 180,E1 -1186.603,E2 -1186.603} C_VEL
LIN {X 0,Y 595.068,Z 330.718,A -85,B 0,C 180,E1 -1186.886,E2 -1186.886} C_VEL
LIN {X 0,Y 595.221,Z 172.552,A -85,B 0,C 180,E1 -1188.851,E2 -1188.851} C_VEL
LIN {X 0,Y 594.71,Z 169.864,A -85,B 0,C 180,E1 -1188.907,E2 -1188.907} C_VEL
LIN {X 0,Y 594.883,Z 145.951,A -85,B 0,C 180,E1 -1191.666,E2 -1191.666} C_VEL
LIN {X 0,Y 595.026,Z 122.541,A -85,B 0,C 180,E1 -1194.418,E2 -1194.418} C_VEL
LIN {X 0,Y 594.986,Z 114.738,A -85,B 0,C 180,E1 -1195.353,E2 -1195.353} C_VEL
LIN {X 0,Y 594.39,Z 112.072,A -85,B 0,C 180,E1 -1195.708,E2 -1195.708} C_VEL
LIN {X 0,Y 594.372,Z 112.077,A -85,B 0,C 180,E1 -1198.227,E2 -1198.227} C_VEL
LIN {X 0,Y 594.381,Z 112.069,A -85,B 0,C 180,E1 -1200.56,E2 -1200.56} C_VEL
LIN {X 0,Y 594.378,Z 112.065,A -85,B 0,C 180,E1 -1202.95,E2 -1202.95} C_VEL
LIN {X 0,Y 594.349,Z 112.072,A -85,B 0,C 180,E1 -1205.409,E2 -1205.409} C_VEL
LIN {X 0,Y 594.383,Z 112.075,A -85,B 0,C 180,E1 -1207.941,E2 -1207.941} C_VEL
LIN {X 0,Y 594.375,Z 112.066,A -85,B 0,C 180,E1 -1210.822,E2 -1210.822} C_VEL
LIN {X 0,Y 594.367,Z 112.071,A -85,B 0,C 180,E1 -1213.3,E2 -1213.3} C_VEL
LIN {X 0,Y 594.368,Z 112.07,A -85,B 0,C 180,E1 -1216.161,E2 -1216.161} C_VEL
LIN {X 0,Y 594.376,Z 112.066,A -85,B 0,C 180,E1 -1218.536,E2 -1218.536} C_VEL
LIN {X 0,Y 594.381,Z 112.072,A -85,B 0,C 180,E1 -1221.296,E2 -1221.296} C_VEL
LIN {X 0,Y 594.349,Z 112.074,A -85,B 0,C 180,E1 -1223.755,E2 -1223.755} C_VEL
LIN {X 0,Y 594.366,Z 112.067,A -85,B 0,C 180,E1 -1226.238,E2 -1226.238} C_VEL
LIN {X 0,Y 594.368,Z 112.069,A -85,B 0,C 180,E1 -1228.65,E2 -1228.65} C_VEL
LIN {X 0,Y 594.384,Z 112.072,A -85,B 0,C 180,E1 -1231.043,E2 -1231.043} C_VEL
LIN {X 0,Y 594.382,Z 112.073,A -85,B 0,C 180,E1 -1233.3,E2 -1233.3} C_VEL
LIN {X 0,Y 594.347,Z 112.072,A -85,B 0,C 180,E1 -1235.576,E2 -1235.576} C_VEL
LIN {X 0,Y 594.36,Z 112.071,A -85,B 0,C 180,E1 -1238.497,E2 -1238.497} C_VEL
LIN {X 0,Y 594.366,Z 112.071,A -85,B 0,C 180,E1 -1241.382,E2 -1241.382} C_VEL
LIN {X 0,Y 594.36,Z 112.069,A -85,B 0,C 180,E1 -1244.219,E2 -1244.219} C_VEL
LIN {X 0,Y 594.374,Z 112.07,A -85,B 0,C 180,E1 -1246.321,E2 -1246.321} C_VEL
LIN {X 0,Y 594.357,Z 112.073,A -85,B 0,C 180,E1 -1249.094,E2 -1249.094} C_VEL
LIN {X 0,Y 594.377,Z 112.066,A -85,B 0,C 180,E1 -1251.843,E2 -1251.843} C_VEL
LIN {X 0,Y 594.388,Z 112.075,A -85,B 0,C 180,E1 -1254.572,E2 -1254.572} C_VEL
LIN {X 0,Y 594.381,Z 112.066,A -85,B 0,C 180,E1 -1257.289,E2 -1257.289} C_VEL
LIN {X 0,Y 594.415,Z 112.065,A -85,B 0,C 180,E1 -1260,E2 -1260} C_VEL
LIN {X 0,Y 594.389,Z 112.069,A -85,B 0,C 180,E1 -1262.711,E2 -1262.711} C_VEL
LIN {X 0,Y 594.372,Z 112.067,A -85,B 0,C 180,E1 -1265.428,E2 -1265.428} C_VEL
LIN {X 0,Y 594.38,Z 112.076,A -85,B 0,C 180,E1 -1268.157,E2 -1268.157} C_VEL
LIN {X 0,Y 594.367,Z 112.067,A -85,B 0,C 180,E1 -1271.061,E2 -1271.061} C_VEL
LIN {X 0,Y 594.372,Z 112.071,A -85,B 0,C 180,E1 -1273.679,E2 -1273.679} C_VEL
LIN {X 0,Y 594.332,Z 112.073,A -85,B 0,C 180,E1 -1275.303,E2 -1275.303} C_VEL
LIN {X 0,Y 593.664,Z 112.164,A -85,B 0,C 180,E1 -1275.869,E2 -1275.869} C_VEL
LIN {X 0,Y 590.801,Z 112.523,A -85,B 0,C 180,E1 -1276.786,E2 -1276.786} C_VEL
LIN {X 0,Y 588.389,Z 112.822,A -85,B 0,C 180,E1 -1277.524,E2 -1277.524} C_VEL
LIN {X 0,Y 587.363,Z 112.947,A -85,B 0,C 180,E1 -1278.094,E2 -1278.094} C_VEL
LIN {X 0,Y 587.285,Z 112.953,A -85,B 0,C 180,E1 -1278.287,E2 -1278.287} C_VEL
LIN {X 0,Y 587.317,Z 112.946,A -85,B 0,C 180,E1 -1281.038,E2 -1281.038} C_VEL
LIN {X 0,Y 587.291,Z 112.954,A -85,B 0,C 180,E1 -1284.009,E2 -1284.009} C_VEL
LIN {X 0,Y 587.302,Z 112.947,A -85,B 0,C 180,E1 -1286.28,E2 -1286.28} C_VEL
LIN {X 0,Y 587.339,Z 112.946,A -85,B 0,C 180,E1 -1289.131,E2 -1289.131} C_VEL
LIN {X 0,Y 587.316,Z 112.951,A -85,B 0,C 180,E1 -1291.831,E2 -1291.831} C_VEL
LIN {X 0,Y 587.327,Z 112.944,A -85,B 0,C 180,E1 -1294.344,E2 -1294.344} C_VEL
LIN {X 0,Y 587.332,Z 112.949,A -85,B 0,C 180,E1 -1297.609,E2 -1297.609} C_VEL
LIN {X 0,Y 587.292,Z 112.948,A -85,B 0,C 180,E1 -1300.256,E2 -1300.256} C_VEL
LIN {X 0,Y 587.287,Z 112.958,A -85,B 0,C 180,E1 -1303.115,E2 -1303.115} C_VEL
LIN {X 0,Y 587.298,Z 112.948,A -85,B 0,C 180,E1 -1306.047,E2 -1306.047} C_VEL
LIN {X 0,Y 587.307,Z 112.956,A -85,B 0,C 180,E1 -1308.928,E2 -1308.928} C_VEL
LIN {X 0,Y 587.3,Z 112.95,A -85,B 0,C 180,E1 -1311.518,E2 -1311.518} C_VEL
LIN {X 0,Y 587.253,Z 112.954,A -85,B 0,C 180,E1 -1314.097,E2 -1314.097} C_VEL
LIN {X 0,Y 587.3,Z 112.955,A -85,B 0,C 180,E1 -1316.601,E2 -1316.601} C_VEL
LIN {X 0,Y 587.285,Z 112.949,A -85,B 0,C 180,E1 -1319.499,E2 -1319.499} C_VEL
LIN {X 0,Y 587.295,Z 112.954,A -85,B 0,C 180,E1 -1322.318,E2 -1322.318} C_VEL
LIN {X 0,Y 587.288,Z 112.953,A -85,B 0,C 180,E1 -1325.238,E2 -1325.238} C_VEL
LIN {X 0,Y 587.329,Z 113.153,A -85,B 0,C 180,E1 -1327.13,E2 -1327.13} C_VEL
LIN {X 0,Y 587.864,Z 117.089,A -85,B 0,C 180,E1 -1327.693,E2 -1327.693} C_VEL
LIN {X 0,Y 587.731,Z 138.345,A -85,B 0,C 180,E1 -1330.575,E2 -1330.575} C_VEL
LIN {X 0,Y 587.689,Z 140.902,A -85,B 0,C 180,E1 -1330.917,E2 -1330.917} C_VEL
LIN {X 0,Y 588.586,Z 145.856,A -85,B 0,C 180,E1 -1331.015,E2 -1331.015} C_VEL
LIN {X 0,Y 588.298,Z 305.975,A -85,B 0,C 180,E1 -1333.037,E2 -1333.037} C_VEL
LIN {X 0,Y 588.226,Z 321.701,A -85,B 0,C 180,E1 -1333.381,E2 -1333.381} C_VEL
LIN {X 0,Y 588.102,Z 337.035,A -85,B 0,C 180,E1 -1333.868,E2 -1333.868} C_VEL
LIN {X 0,Y 587.96,Z 351.703,A -85,B 0,C 180,E1 -1334.487,E2 -1334.487} C_VEL
LIN {X 0,Y 587.842,Z 365.01,A -85,B 0,C 180,E1 -1335.194,E2 -1335.194} C_VEL
LIN {X 0,Y 587.735,Z 378.176,A -85,B 0,C 180,E1 -1336.047,E2 -1336.047} C_VEL
LIN {X 0,Y 587.558,Z 390.866,A -85,B 0,C 180,E1 -1337.04,E2 -1337.04} C_VEL
LIN {X 0,Y 587.472,Z 402.067,A -85,B 0,C 180,E1 -1338.091,E2 -1338.091} C_VEL
LIN {X 0,Y 587.382,Z 412.951,A -85,B 0,C 180,E1 -1339.312,E2 -1339.312} C_VEL
LIN {X 0,Y 587.285,Z 421.994,A -85,B 0,C 180,E1 -1340.529,E2 -1340.529} C_VEL
LIN {X 0,Y 587.258,Z 429.487,A -85,B 0,C 180,E1 -1341.743,E2 -1341.743} C_VEL
LIN {X 0,Y 587.208,Z 436.492,A -85,B 0,C 180,E1 -1343.126,E2 -1343.126} C_VEL
LIN {X 0,Y 587.198,Z 442.001,A -85,B 0,C 180,E1 -1344.506,E2 -1344.506} C_VEL
LIN {X 0,Y 587.169,Z 446.173,A -85,B 0,C 180,E1 -1345.882,E2 -1345.882} C_VEL
LIN {X 0,Y 587.127,Z 449.113,A -85,B 0,C 180,E1 -1347.256,E2 -1347.256} C_VEL
LIN {X 0,Y 587.143,Z 450.88,A -85,B 0,C 180,E1 -1348.628,E2 -1348.628} C_VEL
LIN {X 0,Y 587.135,Z 451.496,A -85,B 0,C 180,E1 -1350,E2 -1350} C_VEL
LIN {X 0,Y 587.145,Z 450.943,A -85,B 0,C 180,E1 -1351.372,E2 -1351.372} C_VEL
LIN {X 0,Y 587.129,Z 449.26,A -85,B 0,C 180,E1 -1352.744,E2 -1352.744} C_VEL
LIN {X 0,Y 587.169,Z 446.406,A -85,B 0,C 180,E1 -1354.118,E2 -1354.118} C_VEL
LIN {X 0,Y 587.198,Z 442.323,A -85,B 0,C 180,E1 -1355.495,E2 -1355.495} C_VEL
LIN {X 0,Y 587.208,Z 436.912,A -85,B 0,C 180,E1 -1356.874,E2 -1356.874} C_VEL
LIN {X 0,Y 587.254,Z 430.012,A -85,B 0,C 180,E1 -1358.257,E2 -1358.257} C_VEL
LIN {X 0,Y 587.287,Z 421.408,A -85,B 0,C 180,E1 -1359.645,E2 -1359.645} C_VEL
LIN {X 0,Y 587.367,Z 412.258,A -85,B 0,C 180,E1 -1360.863,E2 -1360.863} C_VEL
LIN {X 0,Y 587.447,Z 402.929,A -85,B 0,C 180,E1 -1361.91,E2 -1361.91} C_VEL
LIN {X 0,Y 587.589,Z 390.888,A -85,B 0,C 180,E1 -1363.048,E2 -1363.048} C_VEL
LIN {X 0,Y 587.711,Z 377.794,A -85,B 0,C 180,E1 -1364.069,E2 -1364.069} C_VEL
LIN {X 0,Y 587.806,Z 365.035,A -85,B 0,C 180,E1 -1364.896,E2 -1364.896} C_VEL
LIN {X 0,Y 587.958,Z 351.729,A -85,B 0,C 180,E1 -1365.602,E2 -1365.602} C_VEL
LIN {X 0,Y 588.083,Z 337.051,A -85,B 0,C 180,E1 -1366.221,E2 -1366.221} C_VEL
LIN {X 0,Y 588.223,Z 321.361,A -85,B 0,C 180,E1 -1366.718,E2 -1366.718} C_VEL
LIN {X 0,Y 588.286,Z 306.35,A -85,B 0,C 180,E1 -1367.046,E2 -1367.046} C_VEL
LIN {X 0,Y 588.591,Z 145.592,A -85,B 0,C 180,E1 -1369.078,E2 -1369.078} C_VEL
LIN {X 0,Y 587.696,Z 140.862,A -85,B 0,C 180,E1 -1369.178,E2 -1369.178} C_VEL
LIN {X 0,Y 587.841,Z 121.795,A -85,B 0,C 180,E1 -1371.754,E2 -1371.754} C_VEL
LIN {X 0,Y 587.836,Z 116.394,A -85,B 0,C 180,E1 -1372.494,E2 -1372.494} C_VEL
LIN {X 0,Y 587.3,Z 112.953,A -85,B 0,C 180,E1 -1373.021,E2 -1373.021} C_VEL
LIN {X 0,Y 587.298,Z 112.959,A -85,B 0,C 180,E1 -1375.519,E2 -1375.519} C_VEL
LIN {X 0,Y 587.285,Z 112.955,A -85,B 0,C 180,E1 -1377.821,E2 -1377.821} C_VEL
LIN {X 0,Y 587.286,Z 112.95,A -85,B 0,C 180,E1 -1380.501,E2 -1380.501} C_VEL
LIN {X 0,Y 587.3,Z 112.956,A -85,B 0,C 180,E1 -1383.399,E2 -1383.399} C_VEL
LIN {X 0,Y 587.251,Z 112.955,A -85,B 0,C 180,E1 -1385.903,E2 -1385.903} C_VEL
LIN {X 0,Y 587.269,Z 112.954,A -85,B 0,C 180,E1 -1388.484,E2 -1388.484} C_VEL
LIN {X 0,Y 587.297,Z 112.957,A -85,B 0,C 180,E1 -1391.161,E2 -1391.161} C_VEL
LIN {X 0,Y 587.303,Z 112.948,A -85,B 0,C 180,E1 -1394.111,E2 -1394.111} C_VEL
LIN {X 0,Y 587.281,Z 112.957,A -85,B 0,C 180,E1 -1396.99,E2 -1396.99} C_VEL
LIN {X 0,Y 587.291,Z 112.949,A -85,B 0,C 180,E1 -1399.744,E2 -1399.744} C_VEL
LIN {X 0,Y 587.33,Z 112.948,A -85,B 0,C 180,E1 -1402.391,E2 -1402.391} C_VEL
LIN {X 0,Y 587.313,Z 112.946,A -85,B 0,C 180,E1 -1405.777,E2 -1405.777} C_VEL
LIN {X 0,Y 587.317,Z 112.949,A -85,B 0,C 180,E1 -1408.23,E2 -1408.23} C_VEL
LIN {X 0,Y 587.301,Z 112.952,A -85,B 0,C 180,E1 -1410.876,E2 -1410.876} C_VEL
LIN {X 0,Y 587.306,Z 112.949,A -85,B 0,C 180,E1 -1413.83,E2 -1413.83} C_VEL
LIN {X 0,Y 587.291,Z 112.952,A -85,B 0,C 180,E1 -1416.74,E2 -1416.74} C_VEL
LIN {X 0,Y 587.304,Z 112.95,A -85,B 0,C 180,E1 -1419.694,E2 -1419.694} C_VEL
LIN {X 0,Y 587.28,Z 112.955,A -85,B 0,C 180,E1 -1421.872,E2 -1421.872} C_VEL
LIN {X 0,Y 587.302,Z 112.949,A -85,B 0,C 180,E1 -1424.736,E2 -1424.736} C_VEL
LIN {X 0,Y 587.279,Z 112.95,A -85,B 0,C 180,E1 -1426.857,E2 -1426.857} C_VEL
LIN {X 0,Y 587.328,Z 112.95,A -85,B 0,C 180,E1 -1429.66,E2 -1429.66} C_VEL
LIN {X 0,Y 587.315,Z 112.948,A -85,B 0,C 180,E1 -1432.436,E2 -1432.436} C_VEL
LIN {X 0,Y 587.338,Z 112.944,A -85,B 0,C 180,E1 -1435.195,E2 -1435.195} C_VEL
LIN {X 0,Y 587.373,Z 112.945,A -85,B 0,C 180,E1 -1437.943,E2 -1437.943} C_VEL
LIN {X 0,Y 587.384,Z 112.941,A -85,B 0,C 180,E1 -1440,E2 -1440} C_VEL
LIN {X 0,Y 587.348,Z 112.942,A -85,B 0,C 180,E1 -1442.743,E2 -1442.743} C_VEL
LIN {X 0,Y 587.351,Z 112.951,A -85,B 0,C 180,E1 -1445.493,E2 -1445.493} C_VEL
LIN {X 0,Y 587.337,Z 112.943,A -85,B 0,C 180,E1 -1448.256,E2 -1448.256} C_VEL
LIN {X 0,Y 587.353,Z 112.948,A -85,B 0,C 180,E1 -1451.133,E2 -1451.133} C_VEL
LIN {X 0,Y 587.322,Z 112.945,A -85,B 0,C 180,E1 -1454.242,E2 -1454.242} C_VEL
LIN {X 0,Y 587.331,Z 112.949,A -85,B 0,C 180,E1 -1456.807,E2 -1456.807} C_VEL
LIN {X 0,Y 587.308,Z 112.95,A -85,B 0,C 180,E1 -1459.576,E2 -1459.576} C_VEL
LIN {X 0,Y 587.314,Z 112.946,A -85,B 0,C 180,E1 -1461.775,E2 -1461.775} C_VEL
LIN {X 0,Y 587.306,Z 112.955,A -85,B 0,C 180,E1 -1464.761,E2 -1464.761} C_VEL
LIN {X 0,Y 587.34,Z 112.943,A -85,B 0,C 180,E1 -1467.818,E2 -1467.818} C_VEL
LIN {X 0,Y 587.323,Z 112.951,A -85,B 0,C 180,E1 -1470.507,E2 -1470.507} C_VEL
LIN {X 0,Y 587.338,Z 112.946,A -85,B 0,C 180,E1 -1473.111,E2 -1473.111} C_VEL
LIN {X 0,Y 587.29,Z 112.95,A -85,B 0,C 180,E1 -1475.9,E2 -1475.9} C_VEL
LIN {X 0,Y 587.321,Z 112.955,A -85,B 0,C 180,E1 -1478.48,E2 -1478.48} C_VEL
LIN {X 0,Y 587.335,Z 112.944,A -85,B 0,C 180,E1 -1481.157,E2 -1481.157} C_VEL
LIN {X 0,Y 587.328,Z 112.95,A -85,B 0,C 180,E1 -1484.113,E2 -1484.113} C_VEL
LIN {X 0,Y 587.313,Z 112.947,A -85,B 0,C 180,E1 -1486.993,E2 -1486.993} C_VEL
LIN {X 0,Y 587.316,Z 112.948,A -85,B 0,C 180,E1 -1489.745,E2 -1489.745} C_VEL
LIN {X 0,Y 587.345,Z 112.948,A -85,B 0,C 180,E1 -1492.392,E2 -1492.392} C_VEL
LIN {X 0,Y 587.345,Z 112.947,A -85,B 0,C 180,E1 -1495.653,E2 -1495.653} C_VEL
LIN {X 0,Y 587.339,Z 112.949,A -85,B 0,C 180,E1 -1498.231,E2 -1498.231} C_VEL
LIN {X 0,Y 587.349,Z 112.943,A -85,B 0,C 180,E1 -1500.867,E2 -1500.867} C_VEL
LIN {X 0,Y 587.36,Z 112.951,A -85,B 0,C 180,E1 -1503.819,E2 -1503.819} C_VEL
LIN {X 0,Y 587.35,Z 113.044,A -85,B 0,C 180,E1 -1504.103,E2 -1504.103} C_VEL
LIN {X 0,Y 588.257,Z 117.961,A -85,B 0,C 180,E1 -1504.734,E2 -1504.734} C_VEL
LIN {X 0,Y 588.057,Z 142.829,A -85,B 0,C 180,E1 -1507.7,E2 -1507.7} C_VEL
LIN {X 0,Y 587.818,Z 168.485,A -85,B 0,C 180,E1 -1510.703,E2 -1510.703} C_VEL
LIN {X 0,Y 587.815,Z 170.017,A -85,B 0,C 180,E1 -1510.87,E2 -1510.87} C_VEL
LIN {X 0,Y 588.595,Z 174.548,A -85,B 0,C 180,E1 -1510.954,E2 -1510.954} C_VEL
LIN {X 0,Y 588.3,Z 336.369,A -85,B 0,C 180,E1 -1512.999,E2 -1512.999} C_VEL
LIN {X 0,Y 588.208,Z 351.703,A -85,B 0,C 180,E1 -1513.336,E2 -1513.336} C_VEL
LIN {X 0,Y 588.083,Z 367.04,A -85,B 0,C 180,E1 -1513.823,E2 -1513.823} C_VEL
LIN {X 0,Y 587.997,Z 380.765,A -85,B 0,C 180,E1 -1514.399,E2 -1514.399} C_VEL
LIN {X 0,Y 587.829,Z 394.239,A -85,B 0,C 180,E1 -1515.105,E2 -1515.105} C_VEL
LIN {X 0,Y 587.741,Z 407.114,A -85,B 0,C 180,E1 -1515.929,E2 -1515.929} C_VEL
LIN {X 0,Y 587.582,Z 419.287,A -85,B 0,C 180,E1 -1516.864,E2 -1516.864} C_VEL
LIN {X 0,Y 587.454,Z 430.748,A -85,B 0,C 180,E1 -1517.915,E2 -1517.915} C_VEL
LIN {X 0,Y 587.348,Z 440.39,A -85,B 0,C 180,E1 -1518.962,E2 -1518.962} C_VEL
LIN {X 0,Y 587.305,Z 449.856,A -85,B 0,C 180,E1 -1520.182,E2 -1520.182} C_VEL
LIN {X 0,Y 587.265,Z 457.732,A -85,B 0,C 180,E1 -1521.397,E2 -1521.397} C_VEL
LIN {X 0,Y 587.215,Z 465.088,A -85,B 0,C 180,E1 -1522.781,E2 -1522.781} C_VEL
LIN {X 0,Y 587.227,Z 470.923,A -85,B 0,C 180,E1 -1524.161,E2 -1524.161} C_VEL
LIN {X 0,Y 587.136,Z 474.384,A -85,B 0,C 180,E1 -1525.194,E2 -1525.194} C_VEL
LIN {X 0,Y 587.18,Z 477.888,A -85,B 0,C 180,E1 -1526.569,E2 -1526.569} C_VEL
LIN {X 0,Y 587.14,Z 480.193,A -85,B 0,C 180,E1 -1527.942,E2 -1527.942} C_VEL
LIN {X 0,Y 587.135,Z 481.349,A -85,B 0,C 180,E1 -1529.314,E2 -1529.314} C_VEL
LIN {X 0,Y 587.135,Z 481.349,A -85,B 0,C 180,E1 -1530.686,E2 -1530.686} C_VEL
LIN {X 0,Y 587.14,Z 480.192,A -85,B 0,C 180,E1 -1532.058,E2 -1532.058} C_VEL
LIN {X 0,Y 587.18,Z 477.886,A -85,B 0,C 180,E1 -1533.431,E2 -1533.431} C_VEL
LIN {X 0,Y 587.136,Z 474.384,A -85,B 0,C 180,E1 -1534.806,E2 -1534.806} C_VEL
LIN {X 0,Y 587.18,Z 469.608,A -85,B 0,C 180,E1 -1536.184,E2 -1536.184} C_VEL
LIN {X 0,Y 587.23,Z 463.424,A -85,B 0,C 180,E1 -1537.565,E2 -1537.565} C_VEL
LIN {X 0,Y 587.266,Z 455.65,A -85,B 0,C 180,E1 -1538.95,E2 -1538.95} C_VEL
LIN {X 0,Y 587.351,Z 447.369,A -85,B 0,C 180,E1 -1540.166,E2 -1540.166} C_VEL
LIN {X 0,Y 587.4,Z 437.394,A -85,B 0,C 180,E1 -1541.386,E2 -1541.386} C_VEL
LIN {X 0,Y 587.522,Z 427.189,A -85,B 0,C 180,E1 -1542.434,E2 -1542.434} C_VEL
LIN {X 0,Y 587.629,Z 415.018,A -85,B 0,C 180,E1 -1543.487,E2 -1543.487} C_VEL
LIN {X 0,Y 587.774,Z 402.057,A -85,B 0,C 180,E1 -1544.416,E2 -1544.416} C_VEL
LIN {X 0,Y 587.89,Z 387.867,A -85,B 0,C 180,E1 -1545.248,E2 -1545.248} C_VEL
LIN {X 0,Y 588.058,Z 373.795,A -85,B 0,C 180,E1 -1545.91,E2 -1545.91} C_VEL
LIN {X 0,Y 588.175,Z 359.301,A -85,B 0,C 180,E1 -1546.442,E2 -1546.442} C_VEL
LIN {X 0,Y 588.279,Z 344.275,A -85,B 0,C 180,E1 -1546.845,E2 -1546.845} C_VEL
LIN {X 0,Y 588.322,Z 329.073,A -85,B 0,C 180,E1 -1547.11,E2 -1547.11} C_VEL
LIN {X 0,Y 588.503,Z 173.483,A -85,B 0,C 180,E1 -1549.062,E2 -1549.062} C_VEL
LIN {X 0,Y 587.797,Z 169.795,A -85,B 0,C 180,E1 -1549.146,E2 -1549.146} C_VEL
LIN {X 0,Y 588.03,Z 144.391,A -85,B 0,C 180,E1 -1552.116,E2 -1552.116} C_VEL
LIN {X 0,Y 588.241,Z 121.12,A -85,B 0,C 180,E1 -1554.888,E2 -1554.888} C_VEL
LIN {X 0,Y 588.099,Z 116.221,A -85,B 0,C 180,E1 -1555.481,E2 -1555.481} C_VEL
LIN {X 0,Y 587.331,Z 112.953,A -85,B 0,C 180,E1 -1555.924,E2 -1555.924} C_VEL
LIN {X 0,Y 587.32,Z 112.95,A -85,B 0,C 180,E1 -1558.597,E2 -1558.597} C_VEL
LIN {X 0,Y 587.329,Z 112.945,A -85,B 0,C 180,E1 -1560.967,E2 -1560.967} C_VEL
LIN {X 0,Y 587.335,Z 112.944,A -85,B 0,C 180,E1 -1563.397,E2 -1563.397} C_VEL
LIN {X 0,Y 587.291,Z 112.959,A -85,B 0,C 180,E1 -1565.9,E2 -1565.9} C_VEL
LIN {X 0,Y 587.326,Z 112.946,A -85,B 0,C 180,E1 -1568.48,E2 -1568.48} C_VEL
LIN {X 0,Y 587.336,Z 112.945,A -85,B 0,C 180,E1 -1571.157,E2 -1571.157} C_VEL
LIN {X 0,Y 587.313,Z 112.95,A -85,B 0,C 180,E1 -1574.112,E2 -1574.112} C_VEL
LIN {X 0,Y 587.317,Z 112.947,A -85,B 0,C 180,E1 -1576.994,E2 -1576.994} C_VEL
LIN {X 0,Y 587.311,Z 112.953,A -85,B 0,C 180,E1 -1579.745,E2 -1579.745} C_VEL
LIN {X 0,Y 587.344,Z 112.942,A -85,B 0,C 180,E1 -1582.392,E2 -1582.392} C_VEL
LIN {X 0,Y 587.343,Z 112.948,A -85,B 0,C 180,E1 -1585.653,E2 -1585.653} C_VEL
LIN {X 0,Y 587.338,Z 112.943,A -85,B 0,C 180,E1 -1588.231,E2 -1588.231} C_VEL
LIN {X 0,Y 587.349,Z 112.946,A -85,B 0,C 180,E1 -1590.867,E2 -1590.867} C_VEL
LIN {X 0,Y 587.311,Z 112.948,A -85,B 0,C 180,E1 -1593.72,E2 -1593.72} C_VEL
LIN {X 0,Y 587.297,Z 112.948,A -85,B 0,C 180,E1 -1595.992,E2 -1595.992} C_VEL
LIN {X 0,Y 587.334,Z 112.953,A -85,B 0,C 180,E1 -1598.963,E2 -1598.963} C_VEL
LIN {X 0,Y 587.341,Z 112.949,A -85,B 0,C 180,E1 -1601.151,E2 -1601.151} C_VEL
LIN {X 0,Y 587.312,Z 112.946,A -85,B 0,C 180,E1 -1604.025,E2 -1604.025} C_VEL
LIN {X 0,Y 587.351,Z 112.943,A -85,B 0,C 180,E1 -1606.154,E2 -1606.154} C_VEL
LIN {X 0,Y 587.34,Z 112.949,A -85,B 0,C 180,E1 -1608.962,E2 -1608.962} C_VEL
LIN {X 0,Y 587.337,Z 112.942,A -85,B 0,C 180,E1 -1611.744,E2 -1611.744} C_VEL
LIN {X 0,Y 587.353,Z 112.951,A -85,B 0,C 180,E1 -1614.507,E2 -1614.507} C_VEL
LIN {X 0,Y 587.351,Z 112.942,A -85,B 0,C 180,E1 -1617.257,E2 -1617.257} C_VEL
LIN {X 0,Y 587.384,Z 112.941,A -85,B 0,C 180,E1 -1620,E2 -1620} C_VEL
LIN {X 0,Y 587.355,Z 112.944,A -85,B 0,C 180,E1 -1622.743,E2 -1622.743} C_VEL
LIN {X 0,Y 587.342,Z 112.943,A -85,B 0,C 180,E1 -1625.493,E2 -1625.493} C_VEL
LIN {X 0,Y 587.339,Z 112.951,A -85,B 0,C 180,E1 -1628.256,E2 -1628.256} C_VEL
LIN {X 0,Y 587.334,Z 112.944,A -85,B 0,C 180,E1 -1631.124,E2 -1631.124} C_VEL
LIN {X 0,Y 587.343,Z 112.948,A -85,B 0,C 180,E1 -1634.25,E2 -1634.25} C_VEL
LIN {X 0,Y 587.285,Z 112.949,A -85,B 0,C 180,E1 -1636.792,E2 -1636.792} C_VEL
LIN {X 0,Y 587.285,Z 112.953,A -85,B 0,C 180,E1 -1638.287,E2 -1638.287} C_VEL
LIN {X 0,Y 586.645,Z 113.032,A -85,B 0,C 180,E1 -1638.859,E2 -1638.859} C_VEL
LIN {X 0,Y 583.834,Z 113.389,A -85,B 0,C 180,E1 -1639.788,E2 -1639.788} C_VEL
LIN {X 0,Y 581.432,Z 113.686,A -85,B 0,C 180,E1 -1640.535,E2 -1640.535} C_VEL
LIN {X 0,Y 580.376,Z 113.813,A -85,B 0,C 180,E1 -1641.112,E2 -1641.112} C_VEL
LIN {X 0,Y 580.278,Z 113.825,A -85,B 0,C 180,E1 -1641.307,E2 -1641.307} C_VEL
LIN {X 0,Y 580.253,Z 113.833,A -85,B 0,C 180,E1 -1643.559,E2 -1643.559} C_VEL
LIN {X 0,Y 580.263,Z 113.823,A -85,B 0,C 180,E1 -1646.328,E2 -1646.328} C_VEL
LIN {X 0,Y 580.27,Z 113.829,A -85,B 0,C 180,E1 -1649.304,E2 -1649.304} C_VEL
LIN {X 0,Y 580.284,Z 113.823,A -85,B 0,C 180,E1 -1652.202,E2 -1652.202} C_VEL
LIN {X 0,Y 580.274,Z 113.823,A -85,B 0,C 180,E1 -1654.697,E2 -1654.697} C_VEL
LIN {X 0,Y 580.282,Z 113.831,A -85,B 0,C 180,E1 -1657.27,E2 -1657.27} C_VEL
LIN {X 0,Y 580.274,Z 113.823,A -85,B 0,C 180,E1 -1660.268,E2 -1660.268} C_VEL
LIN {X 0,Y 580.249,Z 113.828,A -85,B 0,C 180,E1 -1662.709,E2 -1662.709} C_VEL
LIN {X 0,Y 580.251,Z 113.829,A -85,B 0,C 180,E1 -1665.611,E2 -1665.611} C_VEL
LIN {X 0,Y 580.239,Z 113.828,A -85,B 0,C 180,E1 -1668.227,E2 -1668.227} C_VEL
LIN {X 0,Y 580.259,Z 113.834,A -85,B 0,C 180,E1 -1670.963,E2 -1670.963} C_VEL
LIN {X 0,Y 580.231,Z 113.829,A -85,B 0,C 180,E1 -1673.593,E2 -1673.593} C_VEL
LIN {X 0,Y 580.253,Z 113.827,A -85,B 0,C 180,E1 -1676.141,E2 -1676.141} C_VEL
LIN {X 0,Y 580.238,Z 113.836,A -85,B 0,C 180,E1 -1678.612,E2 -1678.612} C_VEL
LIN {X 0,Y 580.242,Z 113.833,A -85,B 0,C 180,E1 -1681.021,E2 -1681.021} C_VEL
LIN {X 0,Y 580.248,Z 113.828,A -85,B 0,C 180,E1 -1683.675,E2 -1683.675} C_VEL
LIN {X 0,Y 580.237,Z 113.838,A -85,B 0,C 180,E1 -1686.44,E2 -1686.44} C_VEL
LIN {X 0,Y 580.25,Z 113.859,A -85,B 0,C 180,E1 -1686.922,E2 -1686.922} C_VEL
LIN {X 0,Y 580.969,Z 118.444,A -85,B 0,C 180,E1 -1687.601,E2 -1687.601} C_VEL
LIN {X 0,Y 580.82,Z 138.508,A -85,B 0,C 180,E1 -1690.356,E2 -1690.356} C_VEL
LIN {X 0,Y 580.791,Z 140.907,A -85,B 0,C 180,E1 -1690.682,E2 -1690.682} C_VEL
LIN {X 0,Y 581.86,Z 146.365,A -85,B 0,C 180,E1 -1690.793,E2 -1690.793} C_VEL
LIN {X 0,Y 581.514,Z 306.353,A -85,B 0,C 180,E1 -1692.839,E2 -1692.839} C_VEL
LIN {X 0,Y 581.414,Z 321.723,A -85,B 0,C 180,E1 -1693.181,E2 -1693.181} C_VEL
LIN {X 0,Y 581.25,Z 337.048,A -85,B 0,C 180,E1 -1693.673,E2 -1693.673} C_VEL
LIN {X 0,Y 581.101,Z 351.712,A -85,B 0,C 180,E1 -1694.299,E2 -1694.299} C_VEL
LIN {X 0,Y 580.921,Z 365.023,A -85,B 0,C 180,E1 -1695.013,E2 -1695.013} C_VEL
LIN {X 0,Y 580.792,Z 378.372,A -85,B 0,C 180,E1 -1695.89,E2 -1695.89} C_VEL
LIN {X 0,Y 580.593,Z 390.874,A -85,B 0,C 180,E1 -1696.881,E2 -1696.881} C_VEL
LIN {X 0,Y 580.46,Z 402.073,A -85,B 0,C 180,E1 -1697.945,E2 -1697.945} C_VEL
LIN {X 0,Y 580.337,Z 413.113,A -85,B 0,C 180,E1 -1699.201,E2 -1699.201} C_VEL
LIN {X 0,Y 580.239,Z 421.997,A -85,B 0,C 180,E1 -1700.413,E2 -1700.413} C_VEL
LIN {X 0,Y 580.195,Z 429.489,A -85,B 0,C 180,E1 -1701.642,E2 -1701.642} C_VEL
LIN {X 0,Y 580.139,Z 436.494,A -85,B 0,C 180,E1 -1703.042,E2 -1703.042} C_VEL
LIN {X 0,Y 580.127,Z 442.004,A -85,B 0,C 180,E1 -1704.438,E2 -1704.438} C_VEL
LIN {X 0,Y 580.087,Z 446.174,A -85,B 0,C 180,E1 -1705.831,E2 -1705.831} C_VEL
LIN {X 0,Y 580.038,Z 449.113,A -85,B 0,C 180,E1 -1707.222,E2 -1707.222} C_VEL
LIN {X 0,Y 580.043,Z 450.879,A -85,B 0,C 180,E1 -1708.611,E2 -1708.611} C_VEL
LIN {X 0,Y 580.035,Z 451.496,A -85,B 0,C 180,E1 -1710,E2 -1710} C_VEL
LIN {X 0,Y 580.044,Z 450.942,A -85,B 0,C 180,E1 -1711.389,E2 -1711.389} C_VEL
LIN {X 0,Y 580.04,Z 449.26,A -85,B 0,C 180,E1 -1712.778,E2 -1712.778} C_VEL
LIN {X 0,Y 580.087,Z 446.405,A -85,B 0,C 180,E1 -1714.169,E2 -1714.169} C_VEL
LIN {X 0,Y 580.123,Z 442.321,A -85,B 0,C 180,E1 -1715.562,E2 -1715.562} C_VEL
LIN {X 0,Y 580.139,Z 436.909,A -85,B 0,C 180,E1 -1716.958,E2 -1716.958} C_VEL
LIN {X 0,Y 580.19,Z 430.009,A -85,B 0,C 180,E1 -1718.358,E2 -1718.358} C_VEL
LIN {X 0,Y 580.235,Z 421.403,A -85,B 0,C 180,E1 -1719.763,E2 -1719.763} C_VEL
LIN {X 0,Y 580.308,Z 411.832,A -85,B 0,C 180,E1 -1721.046,E2 -1721.046} C_VEL
LIN {X 0,Y 580.463,Z 401.198,A -85,B 0,C 180,E1 -1722.233,E2 -1722.233} C_VEL
LIN {X 0,Y 580.607,Z 389.824,A -85,B 0,C 180,E1 -1723.296,E2 -1723.296} C_VEL
LIN {X 0,Y 580.761,Z 377.061,A -85,B 0,C 180,E1 -1724.292,E2 -1724.292} C_VEL
LIN {X 0,Y 580.94,Z 363.462,A -85,B 0,C 180,E1 -1725.166,E2 -1725.166} C_VEL
LIN {X 0,Y 581.136,Z 349.784,A -85,B 0,C 180,E1 -1725.88,E2 -1725.88} C_VEL
LIN {X 0,Y 581.266,Z 335.789,A -85,B 0,C 180,E1 -1726.462,E2 -1726.462} C_VEL
LIN {X 0,Y 581.447,Z 320.851,A -85,B 0,C 180,E1 -1726.931,E2 -1726.931} C_VEL
LIN {X 0,Y 581.513,Z 306.365,A -85,B 0,C 180,E1 -1727.25,E2 -1727.25} C_VEL
LIN {X 0,Y 581.793,Z 146.148,A -85,B 0,C 180,E1 -1729.302,E2 -1729.302} C_VEL
LIN {X 0,Y 580.787,Z 140.907,A -85,B 0,C 180,E1 -1729.408,E2 -1729.408} C_VEL
LIN {X 0,Y 580.963,Z 121.791,A -85,B 0,C 180,E1 -1732.025,E2 -1732.025} C_VEL
LIN {X 0,Y 580.759,Z 116.426,A -85,B 0,C 180,E1 -1732.783,E2 -1732.783} C_VEL
LIN {X 0,Y 580.252,Z 113.832,A -85,B 0,C 180,E1 -1733.204,E2 -1733.204} C_VEL
LIN {X 0,Y 580.247,Z 113.833,A -85,B 0,C 180,E1 -1735.851,E2 -1735.851} C_VEL
LIN {X 0,Y 580.224,Z 113.831,A -85,B 0,C 180,E1 -1738.19,E2 -1738.19} C_VEL
LIN {X 0,Y 580.239,Z 113.829,A -85,B 0,C 180,E1 -1740.687,E2 -1740.687} C_VEL
LIN {X 0,Y 580.249,Z 113.836,A -85,B 0,C 180,E1 -1743.308,E2 -1743.308} C_VEL
LIN {X 0,Y 580.202,Z 113.835,A -85,B 0,C 180,E1 -1745.75,E2 -1745.75} C_VEL
LIN {X 0,Y 580.233,Z 113.829,A -85,B 0,C 180,E1 -1748.151,E2 -1748.151} C_VEL
LIN {X 0,Y 580.248,Z 113.832,A -85,B 0,C 180,E1 -1750.848,E2 -1750.848} C_VEL
LIN {X 0,Y 580.234,Z 113.829,A -85,B 0,C 180,E1 -1753.662,E2 -1753.662} C_VEL
LIN {X 0,Y 580.228,Z 113.831,A -85,B 0,C 180,E1 -1756.337,E2 -1756.337} C_VEL
LIN {X 0,Y 580.25,Z 113.831,A -85,B 0,C 180,E1 -1759.152,E2 -1759.152} C_VEL
LIN {X 0,Y 580.276,Z 113.822,A -85,B 0,C 180,E1 -1761.929,E2 -1761.929} C_VEL
LIN {X 0,Y 580.215,Z 113.836,A -85,B 0,C 180,E1 -1764.45,E2 -1764.45} C_VEL
LIN {X 0,Y 580.282,Z 113.825,A -85,B 0,C 180,E1 -1766.974,E2 -1766.974} C_VEL
LIN {X 0,Y 580.253,Z 113.824,A -85,B 0,C 180,E1 -1769.422,E2 -1769.422} C_VEL
LIN {X 0,Y 580.241,Z 113.832,A -85,B 0,C 180,E1 -1772.153,E2 -1772.153} C_VEL
LIN {X 0,Y 580.282,Z 113.824,A -85,B 0,C 180,E1 -1774.919,E2 -1774.919} C_VEL
LIN {X 0,Y 580.233,Z 113.832,A -85,B 0,C 180,E1 -1777.946,E2 -1777.946} C_VEL
LIN {X 0,Y 580.279,Z 113.823,A -85,B 0,C 180,E1 -1780.913,E2 -1780.913} C_VEL
LIN {X 0,Y 580.24,Z 113.832,A -85,B 0,C 180,E1 -1783.824,E2 -1783.824} C_VEL
LIN {X 0,Y 580.305,Z 113.828,A -85,B 0,C 180,E1 -1785.982,E2 -1785.982} C_VEL
LIN {X 0,Y 580.31,Z 113.819,A -85,B 0,C 180,E1 -1788.827,E2 -1788.827} C_VEL
LIN {X 0,Y 580.305,Z 113.824,A -85,B 0,C 180,E1 -1791.644,E2 -1791.644} C_VEL
LIN {X 0,Y 580.31,Z 113.819,A -85,B 0,C 180,E1 -1794.44,E2 -1794.44} C_VEL
LIN {X 0,Y 580.343,Z 113.821,A -85,B 0,C 180,E1 -1797.918,E2 -1797.918} C_VEL
LIN {X 0,Y 580.353,Z 113.817,A -85,B 0,C 180,E1 -1800,E2 -1800} C_VEL
LIN {X 0,Y 580.318,Z 113.818,A -85,B 0,C 180,E1 -1802.777,E2 -1802.777} C_VEL
LIN {X 0,Y 580.317,Z 113.827,A -85,B 0,C 180,E1 -1805.56,E2 -1805.56} C_VEL
LIN {X 0,Y 580.306,Z 113.819,A -85,B 0,C 180,E1 -1808.356,E2 -1808.356} C_VEL
LIN {X 0,Y 580.305,Z 113.827,A -85,B 0,C 180,E1 -1811.191,E2 -1811.191} C_VEL
LIN {X 0,Y 580.3,Z 113.82,A -85,B 0,C 180,E1 -1814.017,E2 -1814.017} C_VEL
LIN {X 0,Y 580.293,Z 113.827,A -85,B 0,C 180,E1 -1816.906,E2 -1816.906} C_VEL
LIN {X 0,Y 580.282,Z 113.823,A -85,B 0,C 180,E1 -1819.823,E2 -1819.823} C_VEL
LIN {X 0,Y 580.256,Z 113.825,A -85,B 0,C 180,E1 -1822.053,E2 -1822.053} C_VEL
LIN {X 0,Y 580.285,Z 113.829,A -85,B 0,C 180,E1 -1825.081,E2 -1825.081} C_VEL
LIN {X 0,Y 580.296,Z 113.822,A -85,B 0,C 180,E1 -1828.186,E2 -1828.186} C_VEL
LIN {X 0,Y 580.274,Z 113.832,A -85,B 0,C 180,E1 -1830.692,E2 -1830.692} C_VEL
LIN {X 0,Y 580.285,Z 113.822,A -85,B 0,C 180,E1 -1833.313,E2 -1833.313} C_VEL
LIN {X 0,Y 580.246,Z 113.827,A -85,B 0,C 180,E1 -1835.756,E2 -1835.756} C_VEL
LIN {X 0,Y 580.285,Z 113.825,A -85,B 0,C 180,E1 -1838.147,E2 -1838.147} C_VEL
LIN {X 0,Y 580.297,Z 113.824,A -85,B 0,C 180,E1 -1840.843,E2 -1840.843} C_VEL
LIN {X 0,Y 580.28,Z 113.823,A -85,B 0,C 180,E1 -1843.658,E2 -1843.658} C_VEL
LIN {X 0,Y 580.275,Z 113.828,A -85,B 0,C 180,E1 -1846.61,E2 -1846.61} C_VEL
LIN {X 0,Y 580.299,Z 113.819,A -85,B 0,C 180,E1 -1849.156,E2 -1849.156} C_VEL
LIN {X 0,Y 580.289,Z 113.828,A -85,B 0,C 180,E1 -1851.927,E2 -1851.927} C_VEL
LIN {X 0,Y 580.251,Z 113.83,A -85,B 0,C 180,E1 -1854.452,E2 -1854.452} C_VEL
LIN {X 0,Y 580.29,Z 113.822,A -85,B 0,C 180,E1 -1856.975,E2 -1856.975} C_VEL
LIN {X 0,Y 580.296,Z 113.824,A -85,B 0,C 180,E1 -1859.425,E2 -1859.425} C_VEL
LIN {X 0,Y 580.298,Z 113.828,A -85,B 0,C 180,E1 -1862.141,E2 -1862.141} C_VEL
LIN {X 0,Y 580.341,Z 113.886,A -85,B 0,C 180,E1 -1863.891,E2 -1863.891} C_VEL
LIN {X 0,Y 581.411,Z 119.215,A -85,B 0,C 180,E1 -1864.588,E2 -1864.588} C_VEL
LIN {X 0,Y 581.201,Z 141.269,A -85,B 0,C 180,E1 -1867.235,E2 -1867.235} C_VEL
LIN {X 0,Y 580.958,Z 166.239,A -85,B 0,C 180,E1 -1870.201,E2 -1870.201} C_VEL
LIN {X 0,Y 580.898,Z 169.904,A -85,B 0,C 180,E1 -1870.63,E2 -1870.63} C_VEL
LIN {X 0,Y 581.875,Z 175.732,A -85,B 0,C 180,E1 -1870.741,E2 -1870.741} C_VEL
LIN {X 0,Y 581.53,Z 336.474,A -85,B 0,C 180,E1 -1872.797,E2 -1872.797} C_VEL
LIN {X 0,Y 581.413,Z 351.701,A -85,B 0,C 180,E1 -1873.136,E2 -1873.136} C_VEL
LIN {X 0,Y 581.243,Z 367.037,A -85,B 0,C 180,E1 -1873.628,E2 -1873.628} C_VEL
LIN {X 0,Y 581.133,Z 380.769,A -85,B 0,C 180,E1 -1874.21,E2 -1874.21} C_VEL
LIN {X 0,Y 580.944,Z 394.242,A -85,B 0,C 180,E1 -1874.924,E2 -1874.924} C_VEL
LIN {X 0,Y 580.805,Z 407.479,A -85,B 0,C 180,E1 -1875.783,E2 -1875.783} C_VEL
LIN {X 0,Y 580.608,Z 419.289,A -85,B 0,C 180,E1 -1876.704,E2 -1876.704} C_VEL
LIN {X 0,Y 580.479,Z 430.748,A -85,B 0,C 180,E1 -1877.768,E2 -1877.768} C_VEL
LIN {X 0,Y 580.307,Z 441.454,A -85,B 0,C 180,E1 -1878.954,E2 -1878.954} C_VEL
LIN {X 0,Y 580.268,Z 449.857,A -85,B 0,C 180,E1 -1880.061,E2 -1880.061} C_VEL
LIN {X 0,Y 580.214,Z 457.733,A -85,B 0,C 180,E1 -1881.291,E2 -1881.291} C_VEL
LIN {X 0,Y 580.13,Z 465.089,A -85,B 0,C 180,E1 -1882.692,E2 -1882.692} C_VEL
LIN {X 0,Y 580.132,Z 470.923,A -85,B 0,C 180,E1 -1884.09,E2 -1884.09} C_VEL
LIN {X 0,Y 580.041,Z 474.385,A -85,B 0,C 180,E1 -1885.135,E2 -1885.135} C_VEL
LIN {X 0,Y 580.105,Z 477.889,A -85,B 0,C 180,E1 -1886.527,E2 -1886.527} C_VEL
LIN {X 0,Y 580.039,Z 480.192,A -85,B 0,C 180,E1 -1887.917,E2 -1887.917} C_VEL
LIN {X 0,Y 580.036,Z 481.349,A -85,B 0,C 180,E1 -1889.306,E2 -1889.306} C_VEL
LIN {X 0,Y 580.036,Z 481.349,A -85,B 0,C 180,E1 -1890.694,E2 -1890.694} C_VEL
LIN {X 0,Y 580.039,Z 480.191,A -85,B 0,C 180,E1 -1892.083,E2 -1892.083} C_VEL
LIN {X 0,Y 580.105,Z 477.887,A -85,B 0,C 180,E1 -1893.473,E2 -1893.473} C_VEL
LIN {X 0,Y 580.041,Z 474.385,A -85,B 0,C 180,E1 -1894.865,E2 -1894.865} C_VEL
LIN {X 0,Y 580.093,Z 469.608,A -85,B 0,C 180,E1 -1896.26,E2 -1896.26} C_VEL
LIN {X 0,Y 580.165,Z 463.423,A -85,B 0,C 180,E1 -1897.658,E2 -1897.658} C_VEL
LIN {X 0,Y 580.207,Z 455.648,A -85,B 0,C 180,E1 -1899.06,E2 -1899.06} C_VEL
LIN {X 0,Y 580.308,Z 447.369,A -85,B 0,C 180,E1 -1900.29,E2 -1900.29} C_VEL
LIN {X 0,Y 580.383,Z 437.394,A -85,B 0,C 180,E1 -1901.525,E2 -1901.525} C_VEL
LIN {X 0,Y 580.541,Z 427.188,A -85,B 0,C 180,E1 -1902.586,E2 -1902.586} C_VEL
LIN {X 0,Y 580.677,Z 415.018,A -85,B 0,C 180,E1 -1903.651,E2 -1903.651} C_VEL
LIN {X 0,Y 580.874,Z 401.528,A -85,B 0,C 180,E1 -1904.625,E2 -1904.625} C_VEL
LIN {X 0,Y 581.022,Z 387.87,A -85,B 0,C 180,E1 -1905.433,E2 -1905.433} C_VEL
LIN {X 0,Y 581.212,Z 373.797,A -85,B 0,C 180,E1 -1906.103,E2 -1906.103} C_VEL
LIN {X 0,Y 581.357,Z 359.302,A -85,B 0,C 180,E1 -1906.64,E2 -1906.64} C_VEL
LIN {X 0,Y 581.487,Z 344.055,A -85,B 0,C 180,E1 -1907.052,E2 -1907.052} C_VEL
LIN {X 0,Y 581.552,Z 328.527,A -85,B 0,C 180,E1 -1907.323,E2 -1907.323} C_VEL
LIN {X 0,Y 581.804,Z 174.664,A -85,B 0,C 180,E1 -1909.275,E2 -1909.275} C_VEL
LIN {X 0,Y 580.897,Z 169.774,A -85,B 0,C 180,E1 -1909.385,E2 -1909.385} C_VEL
LIN {X 0,Y 581.199,Z 144.391,A -85,B 0,C 180,E1 -1912.39,E2 -1912.39} C_VEL
LIN {X 0,Y 581.407,Z 120.794,A -85,B 0,C 180,E1 -1915.22,E2 -1915.22} C_VEL
LIN {X 0,Y 581.198,Z 117.63,A -85,B 0,C 180,E1 -1915.614,E2 -1915.614} C_VEL
LIN {X 0,Y 580.315,Z 113.828,A -85,B 0,C 180,E1 -1916.147,E2 -1916.147} C_VEL
LIN {X 0,Y 580.292,Z 113.823,A -85,B 0,C 180,E1 -1918.976,E2 -1918.976} C_VEL
LIN {X 0,Y 580.275,Z 113.825,A -85,B 0,C 180,E1 -1921.386,E2 -1921.386} C_VEL
LIN {X 0,Y 580.315,Z 113.825,A -85,B 0,C 180,E1 -1923.855,E2 -1923.855} C_VEL
LIN {X 0,Y 580.299,Z 113.82,A -85,B 0,C 180,E1 -1926.934,E2 -1926.934} C_VEL
LIN {X 0,Y 580.295,Z 113.829,A -85,B 0,C 180,E1 -1929.933,E2 -1929.933} C_VEL
LIN {X 0,Y 580.277,Z 113.823,A -85,B 0,C 180,E1 -1932.707,E2 -1932.707} C_VEL
LIN {X 0,Y 580.269,Z 113.833,A -85,B 0,C 180,E1 -1935.61,E2 -1935.61} C_VEL
LIN {X 0,Y 580.28,Z 113.824,A -85,B 0,C 180,E1 -1938.231,E2 -1938.231} C_VEL
LIN {X 0,Y 580.278,Z 113.825,A -85,B 0,C 180,E1 -1940.965,E2 -1940.965} C_VEL
LIN {X 0,Y 580.269,Z 113.83,A -85,B 0,C 180,E1 -1943.596,E2 -1943.596} C_VEL
LIN {X 0,Y 580.283,Z 113.822,A -85,B 0,C 180,E1 -1946.143,E2 -1946.143} C_VEL
LIN {X 0,Y 580.272,Z 113.824,A -85,B 0,C 180,E1 -1948.614,E2 -1948.614} C_VEL
LIN {X 0,Y 580.291,Z 113.827,A -85,B 0,C 180,E1 -1951.024,E2 -1951.024} C_VEL
LIN {X 0,Y 580.269,Z 113.826,A -85,B 0,C 180,E1 -1953.671,E2 -1953.671} C_VEL
LIN {X 0,Y 580.257,Z 113.826,A -85,B 0,C 180,E1 -1956.441,E2 -1956.441} C_VEL
LIN {X 0,Y 580.268,Z 113.826,A -85,B 0,C 180,E1 -1959.437,E2 -1959.437} C_VEL
LIN {X 0,Y 580.253,Z 113.827,A -85,B 0,C 180,E1 -1961.645,E2 -1961.645} C_VEL
LIN {X 0,Y 580.261,Z 113.824,A -85,B 0,C 180,E1 -1963.825,E2 -1963.825} C_VEL
LIN {X 0,Y 580.309,Z 113.819,A -85,B 0,C 180,E1 -1965.983,E2 -1965.983} C_VEL
LIN {X 0,Y 580.309,Z 113.827,A -85,B 0,C 180,E1 -1968.827,E2 -1968.827} C_VEL
LIN {X 0,Y 580.307,Z 113.818,A -85,B 0,C 180,E1 -1971.644,E2 -1971.644} C_VEL
LIN {X 0,Y 580.319,Z 113.826,A -85,B 0,C 180,E1 -1974.44,E2 -1974.44} C_VEL
LIN {X 0,Y 580.342,Z 113.817,A -85,B 0,C 180,E1 -1977.918,E2 -1977.918} C_VEL
LIN {X 0,Y 580.353,Z 113.818,A -85,B 0,C 180,E1 -1980.694,E2 -1980.694} C_VEL
LIN {X 0,Y 580.321,Z 113.82,A -85,B 0,C 180,E1 -1982.777,E2 -1982.777} C_VEL
LIN {X 0,Y 580.311,Z 113.819,A -85,B 0,C 180,E1 -1985.56,E2 -1985.56} C_VEL
LIN {X 0,Y 580.307,Z 113.825,A -85,B 0,C 180,E1 -1988.356,E2 -1988.356} C_VEL
LIN {X 0,Y 580.304,Z 113.819,A -85,B 0,C 180,E1 -1991.191,E2 -1991.191} C_VEL
LIN {X 0,Y 580.3,Z 113.825,A -85,B 0,C 180,E1 -1994.331,E2 -1994.331} C_VEL
LIN {X 0,Y 580.234,Z 113.827,A -85,B 0,C 180,E1 -1996.9,E2 -1996.9} C_VEL
LIN {X 0,Y 580.275,Z 113.833,A -85,B 0,C 180,E1 -1999.823,E2 -1999.823} C_VEL
LIN {X 0,Y 580.278,Z 113.825,A -85,B 0,C 180,E1 -2001.307,E2 -2001.307} C_VEL
LIN {X 0,Y 579.571,Z 113.919,A -85,B 0,C 180,E1 -2001.886,E2 -2001.886} C_VEL
LIN {X 0,Y 576.688,Z 114.273,A -85,B 0,C 180,E1 -2002.826,E2 -2002.826} C_VEL
LIN {X 0,Y 574.285,Z 114.577,A -85,B 0,C 180,E1 -2003.582,E2 -2003.582} C_VEL
LIN {X 0,Y 573.273,Z 114.698,A -85,B 0,C 180,E1 -2004.166,E2 -2004.166} C_VEL
LIN {X 0,Y 573.2,Z 114.705,A -85,B 0,C 180,E1 -2004.364,E2 -2004.364} C_VEL
LIN {X 0,Y 573.193,Z 114.703,A -85,B 0,C 180,E1 -2006.979,E2 -2006.979} C_VEL
LIN {X 0,Y 573.215,Z 114.711,A -85,B 0,C 180,E1 -2009.482,E2 -2009.482} C_VEL
LIN {X 0,Y 573.237,Z 114.7,A -85,B 0,C 180,E1 -2012.225,E2 -2012.225} C_VEL
LIN {X 0,Y 573.22,Z 114.702,A -85,B 0,C 180,E1 -2014.769,E2 -2014.769} C_VEL
LIN {X 0,Y 573.221,Z 114.704,A -85,B 0,C 180,E1 -2017.809,E2 -2017.809} C_VEL
LIN {X 0,Y 573.229,Z 114.701,A -85,B 0,C 180,E1 -2020.527,E2 -2020.527} C_VEL
LIN {X 0,Y 573.205,Z 114.706,A -85,B 0,C 180,E1 -2023.665,E2 -2023.665} C_VEL
LIN {X 0,Y 573.198,Z 114.708,A -85,B 0,C 180,E1 -2026.637,E2 -2026.637} C_VEL
LIN {X 0,Y 573.212,Z 114.706,A -85,B 0,C 180,E1 -2029.479,E2 -2029.479} C_VEL
LIN {X 0,Y 573.219,Z 114.703,A -85,B 0,C 180,E1 -2032.191,E2 -2032.191} C_VEL
LIN {X 0,Y 573.208,Z 114.708,A -85,B 0,C 180,E1 -2035.233,E2 -2035.233} C_VEL
LIN {X 0,Y 573.221,Z 114.702,A -85,B 0,C 180,E1 -2037.777,E2 -2037.777} C_VEL
LIN {X 0,Y 573.212,Z 114.708,A -85,B 0,C 180,E1 -2040.631,E2 -2040.631} C_VEL
LIN {X 0,Y 573.193,Z 114.707,A -85,B 0,C 180,E1 -2043.517,E2 -2043.517} C_VEL
LIN {X 0,Y 573.202,Z 114.714,A -85,B 0,C 180,E1 -2046.517,E2 -2046.517} C_VEL
LIN {X 0,Y 573.211,Z 114.761,A -85,B 0,C 180,E1 -2046.728,E2 -2046.728} C_VEL
LIN {X 0,Y 574.104,Z 119.94,A -85,B 0,C 180,E1 -2047.508,E2 -2047.508} C_VEL
LIN {X 0,Y 573.88,Z 139.768,A -85,B 0,C 180,E1 -2050.282,E2 -2050.282} C_VEL
LIN {X 0,Y 573.864,Z 140.918,A -85,B 0,C 180,E1 -2050.44,E2 -2050.44} C_VEL
LIN {X 0,Y 575.156,Z 147.404,A -85,B 0,C 180,E1 -2050.573,E2 -2050.573} C_VEL
LIN {X 0,Y 574.758,Z 305.406,A -85,B 0,C 180,E1 -2052.615,E2 -2052.615} C_VEL
LIN {X 0,Y 574.644,Z 320.88,A -85,B 0,C 180,E1 -2052.954,E2 -2052.954} C_VEL
LIN {X 0,Y 574.457,Z 335.825,A -85,B 0,C 180,E1 -2053.429,E2 -2053.429} C_VEL
LIN {X 0,Y 574.293,Z 349.796,A -85,B 0,C 180,E1 -2054.017,E2 -2054.017} C_VEL
LIN {X 0,Y 574.035,Z 363.47,A -85,B 0,C 180,E1 -2054.738,E2 -2054.738} C_VEL
LIN {X 0,Y 573.864,Z 377.243,A -85,B 0,C 180,E1 -2055.635,E2 -2055.635} C_VEL
LIN {X 0,Y 573.64,Z 389.826,A -85,B 0,C 180,E1 -2056.629,E2 -2056.629} C_VEL
LIN {X 0,Y 573.479,Z 400.304,A -85,B 0,C 180,E1 -2057.616,E2 -2057.616} C_VEL
LIN {X 0,Y 573.335,Z 410.193,A -85,B 0,C 180,E1 -2058.71,E2 -2058.71} C_VEL
LIN {X 0,Y 573.244,Z 419.545,A -85,B 0,C 180,E1 -2059.938,E2 -2059.938} C_VEL
LIN {X 0,Y 573.134,Z 428.484,A -85,B 0,C 180,E1 -2061.361,E2 -2061.361} C_VEL
LIN {X 0,Y 573.075,Z 434.883,A -85,B 0,C 180,E1 -2062.602,E2 -2062.602} C_VEL
LIN {X 0,Y 573.042,Z 440.767,A -85,B 0,C 180,E1 -2064.016,E2 -2064.016} C_VEL
LIN {X 0,Y 572.949,Z 444.251,A -85,B 0,C 180,E1 -2065.074,E2 -2065.074} C_VEL
LIN {X 0,Y 573.004,Z 447.794,A -85,B 0,C 180,E1 -2066.484,E2 -2066.484} C_VEL
LIN {X 0,Y 572.938,Z 450.138,A -85,B 0,C 180,E1 -2067.891,E2 -2067.891} C_VEL
LIN {X 0,Y 572.936,Z 451.337,A -85,B 0,C 180,E1 -2069.297,E2 -2069.297} C_VEL
LIN {X 0,Y 572.937,Z 451.359,A -85,B 0,C 180,E1 -2070.703,E2 -2070.703} C_VEL
LIN {X 0,Y 572.939,Z 450.243,A -85,B 0,C 180,E1 -2072.109,E2 -2072.109} C_VEL
LIN {X 0,Y 573.006,Z 447.982,A -85,B 0,C 180,E1 -2073.516,E2 -2073.516} C_VEL
LIN {X 0,Y 572.949,Z 444.521,A -85,B 0,C 180,E1 -2074.926,E2 -2074.926} C_VEL
LIN {X 0,Y 573.007,Z 439.787,A -85,B 0,C 180,E1 -2076.338,E2 -2076.338} C_VEL
LIN {X 0,Y 573.094,Z 433.653,A -85,B 0,C 180,E1 -2077.753,E2 -2077.753} C_VEL
LIN {X 0,Y 573.134,Z 425.932,A -85,B 0,C 180,E1 -2079.173,E2 -2079.173} C_VEL
LIN {X 0,Y 573.265,Z 417.693,A -85,B 0,C 180,E1 -2080.418,E2 -2080.418} C_VEL
LIN {X 0,Y 573.38,Z 407.784,A -85,B 0,C 180,E1 -2081.668,E2 -2081.668} C_VEL
LIN {X 0,Y 573.534,Z 397.631,A -85,B 0,C 180,E1 -2082.743,E2 -2082.743} C_VEL
LIN {X 0,Y 573.722,Z 385.55,A -85,B 0,C 180,E1 -2083.82,E2 -2083.82} C_VEL
LIN {X 0,Y 573.937,Z 372.592,A -85,B 0,C 180,E1 -2084.78,E2 -2084.78} C_VEL
LIN {X 0,Y 574.122,Z 358.713,A -85,B 0,C 180,E1 -2085.623,E2 -2085.623} C_VEL
LIN {X 0,Y 574.353,Z 343.781,A -85,B 0,C 180,E1 -2086.346,E2 -2086.346} C_VEL
LIN {X 0,Y 574.544,Z 329.264,A -85,B 0,C 180,E1 -2086.889,E2 -2086.889} C_VEL
LIN {X 0,Y 574.687,Z 313.683,A -85,B 0,C 180,E1 -2087.314,E2 -2087.314} C_VEL
LIN {X 0,Y 574.779,Z 298.74,A -85,B 0,C 180,E1 -2087.576,E2 -2087.576} C_VEL
LIN {X 0,Y 575.094,Z 147.17,A -85,B 0,C 180,E1 -2089.522,E2 -2089.522} C_VEL
LIN {X 0,Y 573.831,Z 140.872,A -85,B 0,C 180,E1 -2089.657,E2 -2089.657} C_VEL
LIN {X 0,Y 574.082,Z 121.929,A -85,B 0,C 180,E1 -2092.303,E2 -2092.303} C_VEL
LIN {X 0,Y 573.88,Z 117.929,A -85,B 0,C 180,E1 -2092.882,E2 -2092.882} C_VEL
LIN {X 0,Y 573.211,Z 114.71,A -85,B 0,C 180,E1 -2093.377,E2 -2093.377} C_VEL
LIN {X 0,Y 573.23,Z 114.704,A -85,B 0,C 180,E1 -2096.192,E2 -2096.192} C_VEL
LIN {X 0,Y 573.177,Z 114.709,A -85,B 0,C 180,E1 -2098.568,E2 -2098.568} C_VEL
LIN {X 0,Y 573.199,Z 114.71,A -85,B 0,C 180,E1 -2100.995,E2 -2100.995} C_VEL
LIN {X 0,Y 573.216,Z 114.709,A -85,B 0,C 180,E1 -2103.517,E2 -2103.517} C_VEL
LIN {X 0,Y 573.176,Z 114.708,A -85,B 0,C 180,E1 -2106.055,E2 -2106.055} C_VEL
LIN {X 0,Y 573.175,Z 114.712,A -85,B 0,C 180,E1 -2108.707,E2 -2108.707} C_VEL
LIN {X 0,Y 573.191,Z 114.708,A -85,B 0,C 180,E1 -2111.588,E2 -2111.588} C_VEL
LIN {X 0,Y 573.209,Z 114.709,A -85,B 0,C 180,E1 -2114.673,E2 -2114.673} C_VEL
LIN {X 0,Y 573.202,Z 114.703,A -85,B 0,C 180,E1 -2117.596,E2 -2117.596} C_VEL
LIN {X 0,Y 573.231,Z 114.707,A -85,B 0,C 180,E1 -2120.57,E2 -2120.57} C_VEL
LIN {X 0,Y 573.228,Z 114.704,A -85,B 0,C 180,E1 -2123.076,E2 -2123.076} C_VEL
LIN {X 0,Y 573.242,Z 114.699,A -85,B 0,C 180,E1 -2125.67,E2 -2125.67} C_VEL
LIN {X 0,Y 573.22,Z 114.704,A -85,B 0,C 180,E1 -2128.183,E2 -2128.183} C_VEL
LIN {X 0,Y 573.217,Z 114.71,A -85,B 0,C 180,E1 -2130.631,E2 -2130.631} C_VEL
LIN {X 0,Y 573.204,Z 114.704,A -85,B 0,C 180,E1 -2133.515,E2 -2133.515} C_VEL
LIN {X 0,Y 573.196,Z 114.711,A -85,B 0,C 180,E1 -2136.133,E2 -2136.133} C_VEL
LIN {X 0,Y 573.229,Z 114.701,A -85,B 0,C 180,E1 -2139.173,E2 -2139.173} C_VEL
LIN {X 0,Y 573.197,Z 114.705,A -85,B 0,C 180,E1 -2141.41,E2 -2141.41} C_VEL
LIN {X 0,Y 573.208,Z 114.709,A -85,B 0,C 180,E1 -2144.351,E2 -2144.351} C_VEL
LIN {X 0,Y 573.204,Z 114.706,A -85,B 0,C 180,E1 -2146.529,E2 -2146.529} C_VEL
LIN {X 0,Y 573.26,Z 114.699,A -85,B 0,C 180,E1 -2149.403,E2 -2149.403} C_VEL
LIN {X 0,Y 573.225,Z 114.705,A -85,B 0,C 180,E1 -2152.249,E2 -2152.249} C_VEL
LIN {X 0,Y 573.287,Z 114.694,A -85,B 0,C 180,E1 -2155.077,E2 -2155.077} C_VEL
LIN {X 0,Y 573.312,Z 114.697,A -85,B 0,C 180,E1 -2157.892,E2 -2157.892} C_VEL
LIN {X 0,Y 573.321,Z 114.693,A -85,B 0,C 180,E1 -2160,E2 -2160} C_VEL
LIN {X 0,Y 573.287,Z 114.694,A -85,B 0,C 180,E1 -2162.811,E2 -2162.811} C_VEL
LIN {X 0,Y 573.284,Z 114.701,A -85,B 0,C 180,E1 -2165.628,E2 -2165.628} C_VEL
LIN {X 0,Y 573.25,Z 114.698,A -85,B 0,C 180,E1 -2168.46,E2 -2168.46} C_VEL
LIN {X 0,Y 573.276,Z 114.705,A -85,B 0,C 180,E1 -2171.312,E2 -2171.312} C_VEL
LIN {X 0,Y 573.258,Z 114.697,A -85,B 0,C 180,E1 -2174.413,E2 -2174.413} C_VEL
LIN {X 0,Y 573.25,Z 114.708,A -85,B 0,C 180,E1 -2177.112,E2 -2177.112} C_VEL
LIN {X 0,Y 573.238,Z 114.7,A -85,B 0,C 180,E1 -2180.077,E2 -2180.077} C_VEL
LIN {X 0,Y 573.224,Z 114.702,A -85,B 0,C 180,E1 -2182.338,E2 -2182.338} C_VEL
LIN {X 0,Y 573.233,Z 114.702,A -85,B 0,C 180,E1 -2185.411,E2 -2185.411} C_VEL
LIN {X 0,Y 573.235,Z 114.706,A -85,B 0,C 180,E1 -2188.564,E2 -2188.564} C_VEL
LIN {X 0,Y 573.221,Z 114.708,A -85,B 0,C 180,E1 -2190.994,E2 -2190.994} C_VEL
LIN {X 0,Y 573.243,Z 114.698,A -85,B 0,C 180,E1 -2193.52,E2 -2193.52} C_VEL
LIN {X 0,Y 573.216,Z 114.705,A -85,B 0,C 180,E1 -2196.051,E2 -2196.051} C_VEL
LIN {X 0,Y 573.239,Z 114.706,A -85,B 0,C 180,E1 -2198.702,E2 -2198.702} C_VEL
LIN {X 0,Y 573.23,Z 114.701,A -85,B 0,C 180,E1 -2201.592,E2 -2201.592} C_VEL
LIN {X 0,Y 573.235,Z 114.71,A -85,B 0,C 180,E1 -2204.333,E2 -2204.333} C_VEL
LIN {X 0,Y 573.241,Z 114.699,A -85,B 0,C 180,E1 -2207.358,E2 -2207.358} C_VEL
LIN {X 0,Y 573.252,Z 114.702,A -85,B 0,C 180,E1 -2210.567,E2 -2210.567} C_VEL
LIN {X 0,Y 573.253,Z 114.698,A -85,B 0,C 180,E1 -2213.077,E2 -2213.077} C_VEL
LIN {X 0,Y 573.266,Z 114.701,A -85,B 0,C 180,E1 -2215.671,E2 -2215.671} C_VEL
LIN {X 0,Y 573.24,Z 114.706,A -85,B 0,C 180,E1 -2218.184,E2 -2218.184} C_VEL
LIN {X 0,Y 573.265,Z 114.699,A -85,B 0,C 180,E1 -2220.634,E2 -2220.634} C_VEL
LIN {X 0,Y 573.251,Z 114.702,A -85,B 0,C 180,E1 -2223.024,E2 -2223.024} C_VEL
LIN {X 0,Y 573.274,Z 114.774,A -85,B 0,C 180,E1 -2223.679,E2 -2223.679} C_VEL
LIN {X 0,Y 574.549,Z 120.61,A -85,B 0,C 180,E1 -2224.457,E2 -2224.457} C_VEL
LIN {X 0,Y 574.373,Z 141.123,A -85,B 0,C 180,E1 -2226.949,E2 -2226.949} C_VEL
LIN {X 0,Y 574.05,Z 166.239,A -85,B 0,C 180,E1 -2229.952,E2 -2229.952} C_VEL
LIN {X 0,Y 574.002,Z 169.853,A -85,B 0,C 180,E1 -2230.382,E2 -2230.382} C_VEL
LIN {X 0,Y 575.174,Z 176.433,A -85,B 0,C 180,E1 -2230.516,E2 -2230.516} C_VEL
LIN {X 0,Y 574.764,Z 336.001,A -85,B 0,C 180,E1 -2232.58,E2 -2232.58} C_VEL
LIN {X 0,Y 574.627,Z 351.699,A -85,B 0,C 180,E1 -2232.93,E2 -2232.93} C_VEL
LIN {X 0,Y 574.442,Z 367.035,A -85,B 0,C 180,E1 -2233.428,E2 -2233.428} C_VEL
LIN {X 0,Y 574.299,Z 380.772,A -85,B 0,C 180,E1 -2234.017,E2 -2234.017} C_VEL
LIN {X 0,Y 574.05,Z 394.246,A -85,B 0,C 180,E1 -2234.739,E2 -2234.739} C_VEL
LIN {X 0,Y 573.861,Z 407.818,A -85,B 0,C 180,E1 -2235.631,E2 -2235.631} C_VEL
LIN {X 0,Y 573.635,Z 420.35,A -85,B 0,C 180,E1 -2236.629,E2 -2236.629} C_VEL
LIN {X 0,Y 573.477,Z 430.748,A -85,B 0,C 180,E1 -2237.616,E2 -2237.616} C_VEL
LIN {X 0,Y 573.286,Z 440.769,A -85,B 0,C 180,E1 -2238.734,E2 -2238.734} C_VEL
LIN {X 0,Y 573.243,Z 449.856,A -85,B 0,C 180,E1 -2239.938,E2 -2239.938} C_VEL
LIN {X 0,Y 573.133,Z 457.734,A -85,B 0,C 180,E1 -2241.183,E2 -2241.183} C_VEL
LIN {X 0,Y 573.074,Z 465.089,A -85,B 0,C 180,E1 -2242.601,E2 -2242.601} C_VEL
LIN {X 0,Y 573.042,Z 470.922,A -85,B 0,C 180,E1 -2244.016,E2 -2244.016} C_VEL
LIN {X 0,Y 572.951,Z 474.385,A -85,B 0,C 180,E1 -2245.074,E2 -2245.074} C_VEL
LIN {X 0,Y 573.005,Z 477.89,A -85,B 0,C 180,E1 -2246.484,E2 -2246.484} C_VEL
LIN {X 0,Y 572.938,Z 480.192,A -85,B 0,C 180,E1 -2247.891,E2 -2247.891} C_VEL
LIN {X 0,Y 572.936,Z 481.349,A -85,B 0,C 180,E1 -2249.297,E2 -2249.297} C_VEL
LIN {X 0,Y 572.936,Z 481.348,A -85,B 0,C 180,E1 -2250.703,E2 -2250.703} C_VEL
LIN {X 0,Y 572.938,Z 480.19,A -85,B 0,C 180,E1 -2252.109,E2 -2252.109} C_VEL
LIN {X 0,Y 573.005,Z 477.887,A -85,B 0,C 180,E1 -2253.516,E2 -2253.516} C_VEL
LIN {X 0,Y 572.951,Z 474.386,A -85,B 0,C 180,E1 -2254.926,E2 -2254.926} C_VEL
LIN {X 0,Y 573.014,Z 469.609,A -85,B 0,C 180,E1 -2256.337,E2 -2256.337} C_VEL
LIN {X 0,Y 573.093,Z 463.422,A -85,B 0,C 180,E1 -2257.753,E2 -2257.753} C_VEL
LIN {X 0,Y 573.135,Z 455.647,A -85,B 0,C 180,E1 -2259.173,E2 -2259.173} C_VEL
LIN {X 0,Y 573.27,Z 447.368,A -85,B 0,C 180,E1 -2260.418,E2 -2260.418} C_VEL
